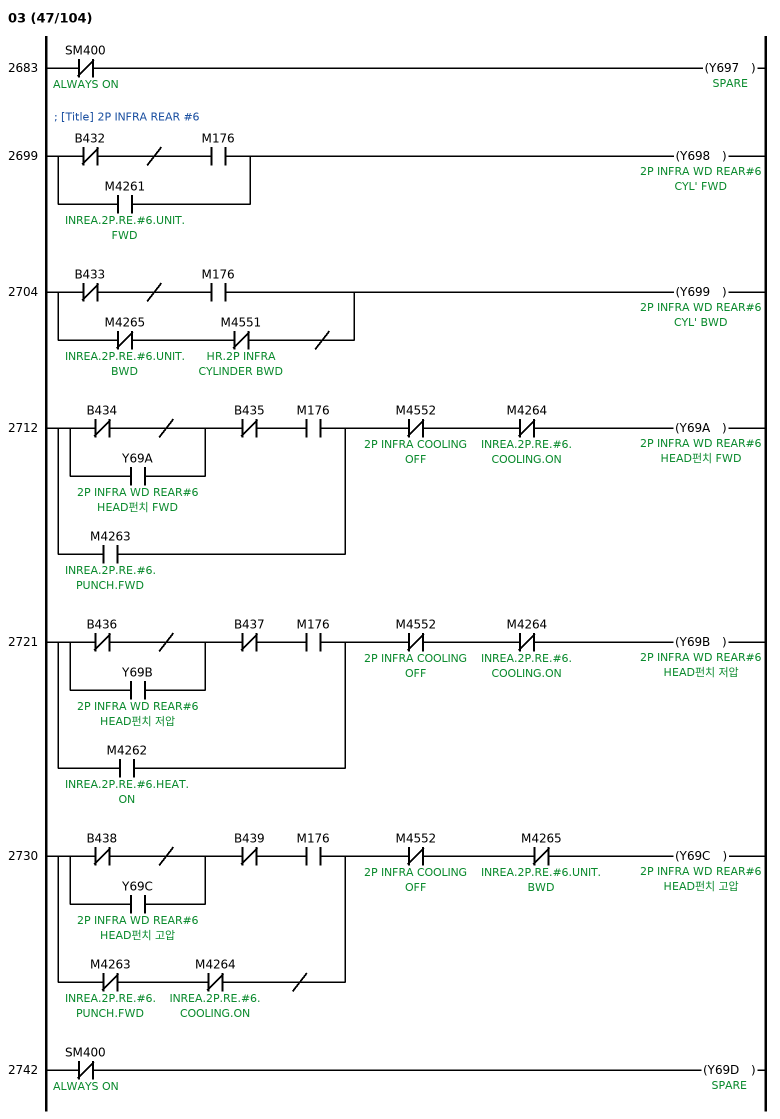
2683  LDI     SM400  ; ALWAYS ON
      OUT     Y697  ; SPARE
; [Title] 2P INFRA REAR #6
2699  LDI     B432
      INV
      AND     M176
      OR      M4261  ; INREA.2P.RE.#6.UNIT.FWD
      OUT     Y698  ; 2P INFRA WD REAR#6 CYL' FWD
2704  LDI     B433
      INV
      AND     M176
      LDI     M4265  ; INREA.2P.RE.#6.UNIT.BWD
      ANI     M4551  ; HR.2P INFRA CYLINDER BWD
      INV
      ORB
      OUT     Y699  ; 2P INFRA WD REAR#6 CYL' BWD
2712  LDI     B434
      INV
      OR      Y69A  ; 2P INFRA WD REAR#6 HEAD펀치 FWD
      ANI     B435
      AND     M176
      OR      M4263  ; INREA.2P.RE.#6.PUNCH.FWD
      ANI     M4552  ; 2P INFRA COOLING OFF
      ANI     M4264  ; INREA.2P.RE.#6.COOLING.ON
      OUT     Y69A  ; 2P INFRA WD REAR#6 HEAD펀치 FWD
2721  LDI     B436
      INV
      OR      Y69B  ; 2P INFRA WD REAR#6 HEAD펀치 저압
      ANI     B437
      AND     M176
      OR      M4262  ; INREA.2P.RE.#6.HEAT.ON
      ANI     M4552  ; 2P INFRA COOLING OFF
      ANI     M4264  ; INREA.2P.RE.#6.COOLING.ON
      OUT     Y69B  ; 2P INFRA WD REAR#6 HEAD펀치 저압
2730  LDI     B438
      INV
      OR      Y69C  ; 2P INFRA WD REAR#6 HEAD펀치 고압
      ANI     B439
      AND     M176
      LDI     M4263  ; INREA.2P.RE.#6.PUNCH.FWD
      ANI     M4264  ; INREA.2P.RE.#6.COOLING.ON
      INV
      ORB
      ANI     M4552  ; 2P INFRA COOLING OFF
      ANI     M4265  ; INREA.2P.RE.#6.UNIT.BWD
      OUT     Y69C  ; 2P INFRA WD REAR#6 HEAD펀치 고압
2742  LDI     SM400  ; ALWAYS ON
      OUT     Y69D  ; SPARE
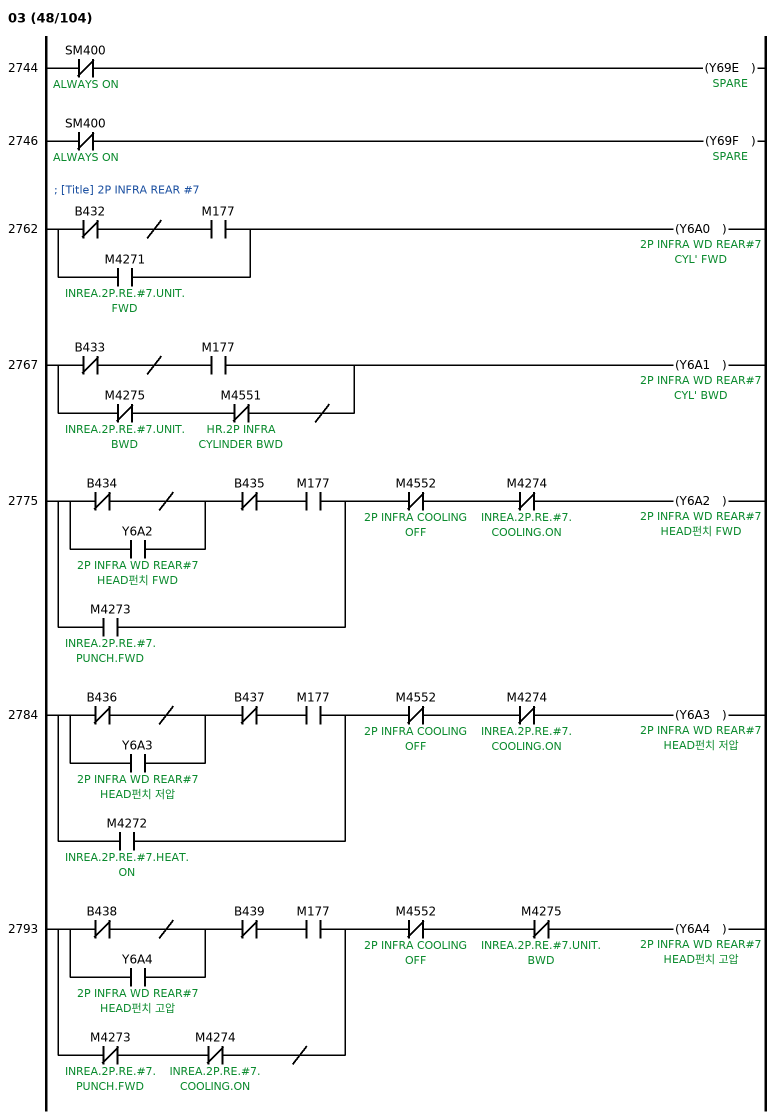
2744  LDI     SM400  ; ALWAYS ON
      OUT     Y69E  ; SPARE
2746  LDI     SM400  ; ALWAYS ON
      OUT     Y69F  ; SPARE
; [Title] 2P INFRA REAR #7
2762  LDI     B432
      INV
      AND     M177
      OR      M4271  ; INREA.2P.RE.#7.UNIT.FWD
      OUT     Y6A0  ; 2P INFRA WD REAR#7 CYL' FWD
2767  LDI     B433
      INV
      AND     M177
      LDI     M4275  ; INREA.2P.RE.#7.UNIT.BWD
      ANI     M4551  ; HR.2P INFRA CYLINDER BWD
      INV
      ORB
      OUT     Y6A1  ; 2P INFRA WD REAR#7 CYL' BWD
2775  LDI     B434
      INV
      OR      Y6A2  ; 2P INFRA WD REAR#7 HEAD펀치 FWD
      ANI     B435
      AND     M177
      OR      M4273  ; INREA.2P.RE.#7.PUNCH.FWD
      ANI     M4552  ; 2P INFRA COOLING OFF
      ANI     M4274  ; INREA.2P.RE.#7.COOLING.ON
      OUT     Y6A2  ; 2P INFRA WD REAR#7 HEAD펀치 FWD
2784  LDI     B436
      INV
      OR      Y6A3  ; 2P INFRA WD REAR#7 HEAD펀치 저압
      ANI     B437
      AND     M177
      OR      M4272  ; INREA.2P.RE.#7.HEAT.ON
      ANI     M4552  ; 2P INFRA COOLING OFF
      ANI     M4274  ; INREA.2P.RE.#7.COOLING.ON
      OUT     Y6A3  ; 2P INFRA WD REAR#7 HEAD펀치 저압
2793  LDI     B438
      INV
      OR      Y6A4  ; 2P INFRA WD REAR#7 HEAD펀치 고압
      ANI     B439
      AND     M177
      LDI     M4273  ; INREA.2P.RE.#7.PUNCH.FWD
      ANI     M4274  ; INREA.2P.RE.#7.COOLING.ON
      INV
      ORB
      ANI     M4552  ; 2P INFRA COOLING OFF
      ANI     M4275  ; INREA.2P.RE.#7.UNIT.BWD
      OUT     Y6A4  ; 2P INFRA WD REAR#7 HEAD펀치 고압
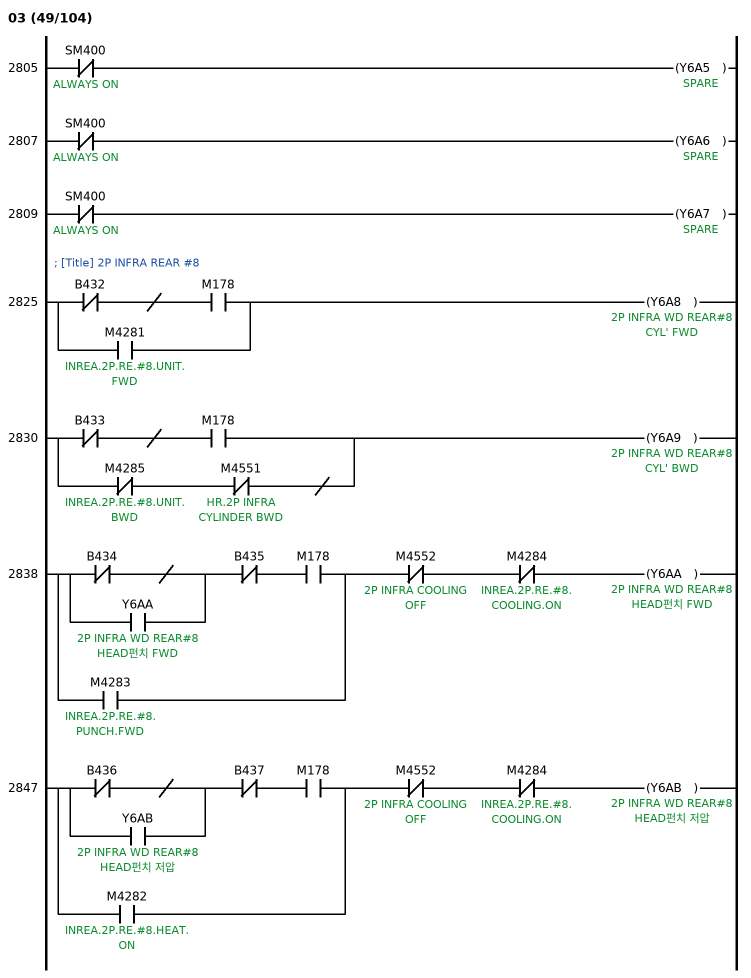
2805  LDI     SM400  ; ALWAYS ON
      OUT     Y6A5  ; SPARE
2807  LDI     SM400  ; ALWAYS ON
      OUT     Y6A6  ; SPARE
2809  LDI     SM400  ; ALWAYS ON
      OUT     Y6A7  ; SPARE
; [Title] 2P INFRA REAR #8
2825  LDI     B432
      INV
      AND     M178
      OR      M4281  ; INREA.2P.RE.#8.UNIT.FWD
      OUT     Y6A8  ; 2P INFRA WD REAR#8 CYL' FWD
2830  LDI     B433
      INV
      AND     M178
      LDI     M4285  ; INREA.2P.RE.#8.UNIT.BWD
      ANI     M4551  ; HR.2P INFRA CYLINDER BWD
      INV
      ORB
      OUT     Y6A9  ; 2P INFRA WD REAR#8 CYL' BWD
2838  LDI     B434
      INV
      OR      Y6AA  ; 2P INFRA WD REAR#8 HEAD펀치 FWD
      ANI     B435
      AND     M178
      OR      M4283  ; INREA.2P.RE.#8.PUNCH.FWD
      ANI     M4552  ; 2P INFRA COOLING OFF
      ANI     M4284  ; INREA.2P.RE.#8.COOLING.ON
      OUT     Y6AA  ; 2P INFRA WD REAR#8 HEAD펀치 FWD
2847  LDI     B436
      INV
      OR      Y6AB  ; 2P INFRA WD REAR#8 HEAD펀치 저압
      ANI     B437
      AND     M178
      OR      M4282  ; INREA.2P.RE.#8.HEAT.ON
      ANI     M4552  ; 2P INFRA COOLING OFF
      ANI     M4284  ; INREA.2P.RE.#8.COOLING.ON
      OUT     Y6AB  ; 2P INFRA WD REAR#8 HEAD펀치 저압
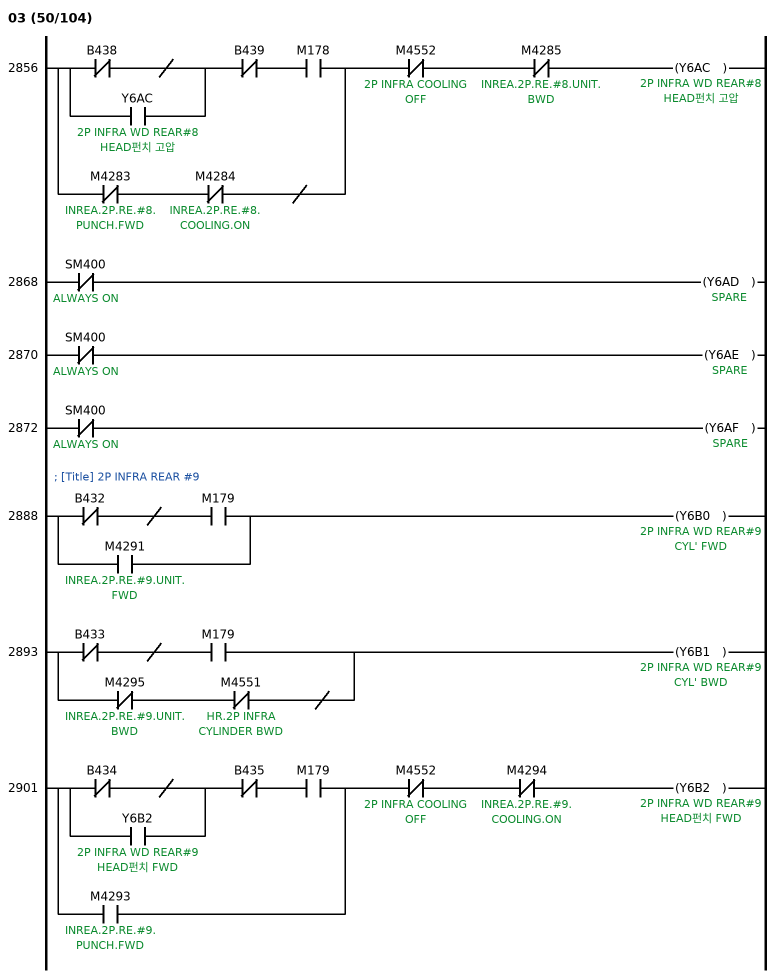
2856  LDI     B438
      INV
      OR      Y6AC  ; 2P INFRA WD REAR#8 HEAD펀치 고압
      ANI     B439
      AND     M178
      LDI     M4283  ; INREA.2P.RE.#8.PUNCH.FWD
      ANI     M4284  ; INREA.2P.RE.#8.COOLING.ON
      INV
      ORB
      ANI     M4552  ; 2P INFRA COOLING OFF
      ANI     M4285  ; INREA.2P.RE.#8.UNIT.BWD
      OUT     Y6AC  ; 2P INFRA WD REAR#8 HEAD펀치 고압
2868  LDI     SM400  ; ALWAYS ON
      OUT     Y6AD  ; SPARE
2870  LDI     SM400  ; ALWAYS ON
      OUT     Y6AE  ; SPARE
2872  LDI     SM400  ; ALWAYS ON
      OUT     Y6AF  ; SPARE
; [Title] 2P INFRA REAR #9
2888  LDI     B432
      INV
      AND     M179
      OR      M4291  ; INREA.2P.RE.#9.UNIT.FWD
      OUT     Y6B0  ; 2P INFRA WD REAR#9 CYL' FWD
2893  LDI     B433
      INV
      AND     M179
      LDI     M4295  ; INREA.2P.RE.#9.UNIT.BWD
      ANI     M4551  ; HR.2P INFRA CYLINDER BWD
      INV
      ORB
      OUT     Y6B1  ; 2P INFRA WD REAR#9 CYL' BWD
2901  LDI     B434
      INV
      OR      Y6B2  ; 2P INFRA WD REAR#9 HEAD펀치 FWD
      ANI     B435
      AND     M179
      OR      M4293  ; INREA.2P.RE.#9.PUNCH.FWD
      ANI     M4552  ; 2P INFRA COOLING OFF
      ANI     M4294  ; INREA.2P.RE.#9.COOLING.ON
      OUT     Y6B2  ; 2P INFRA WD REAR#9 HEAD펀치 FWD
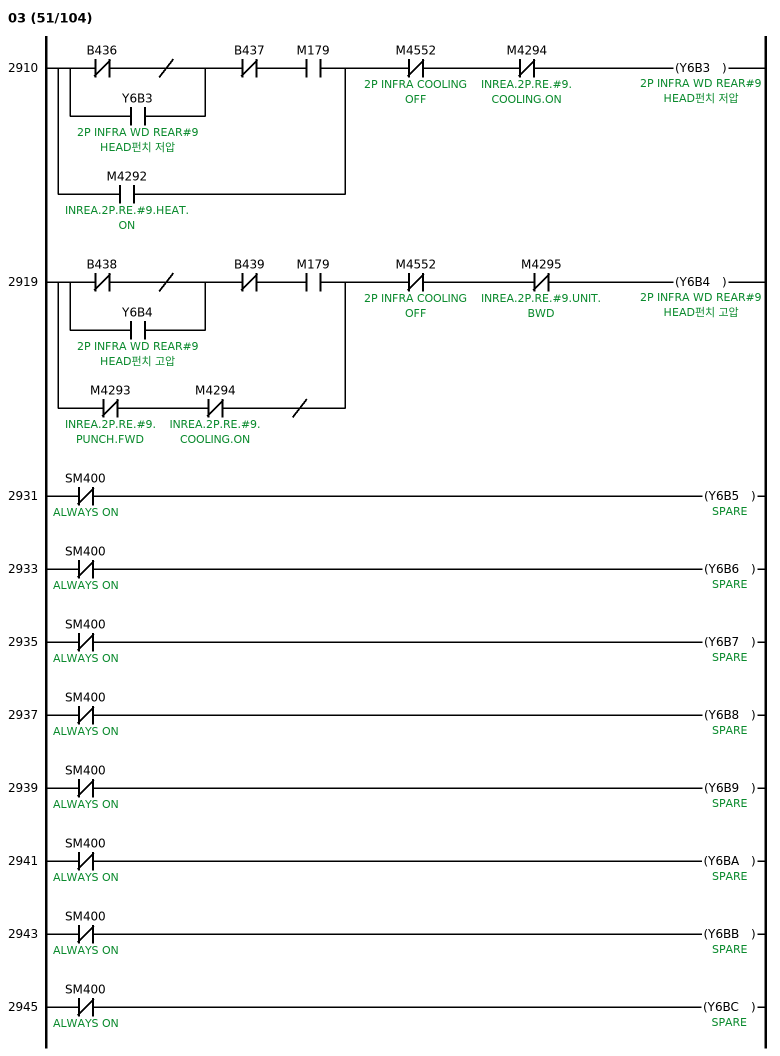
2910  LDI     B436
      INV
      OR      Y6B3  ; 2P INFRA WD REAR#9 HEAD펀치 저압
      ANI     B437
      AND     M179
      OR      M4292  ; INREA.2P.RE.#9.HEAT.ON
      ANI     M4552  ; 2P INFRA COOLING OFF
      ANI     M4294  ; INREA.2P.RE.#9.COOLING.ON
      OUT     Y6B3  ; 2P INFRA WD REAR#9 HEAD펀치 저압
2919  LDI     B438
      INV
      OR      Y6B4  ; 2P INFRA WD REAR#9 HEAD펀치 고압
      ANI     B439
      AND     M179
      LDI     M4293  ; INREA.2P.RE.#9.PUNCH.FWD
      ANI     M4294  ; INREA.2P.RE.#9.COOLING.ON
      INV
      ORB
      ANI     M4552  ; 2P INFRA COOLING OFF
      ANI     M4295  ; INREA.2P.RE.#9.UNIT.BWD
      OUT     Y6B4  ; 2P INFRA WD REAR#9 HEAD펀치 고압
2931  LDI     SM400  ; ALWAYS ON
      OUT     Y6B5  ; SPARE
2933  LDI     SM400  ; ALWAYS ON
      OUT     Y6B6  ; SPARE
2935  LDI     SM400  ; ALWAYS ON
      OUT     Y6B7  ; SPARE
2937  LDI     SM400  ; ALWAYS ON
      OUT     Y6B8  ; SPARE
2939  LDI     SM400  ; ALWAYS ON
      OUT     Y6B9  ; SPARE
2941  LDI     SM400  ; ALWAYS ON
      OUT     Y6BA  ; SPARE
2943  LDI     SM400  ; ALWAYS ON
      OUT     Y6BB  ; SPARE
2945  LDI     SM400  ; ALWAYS ON
      OUT     Y6BC  ; SPARE
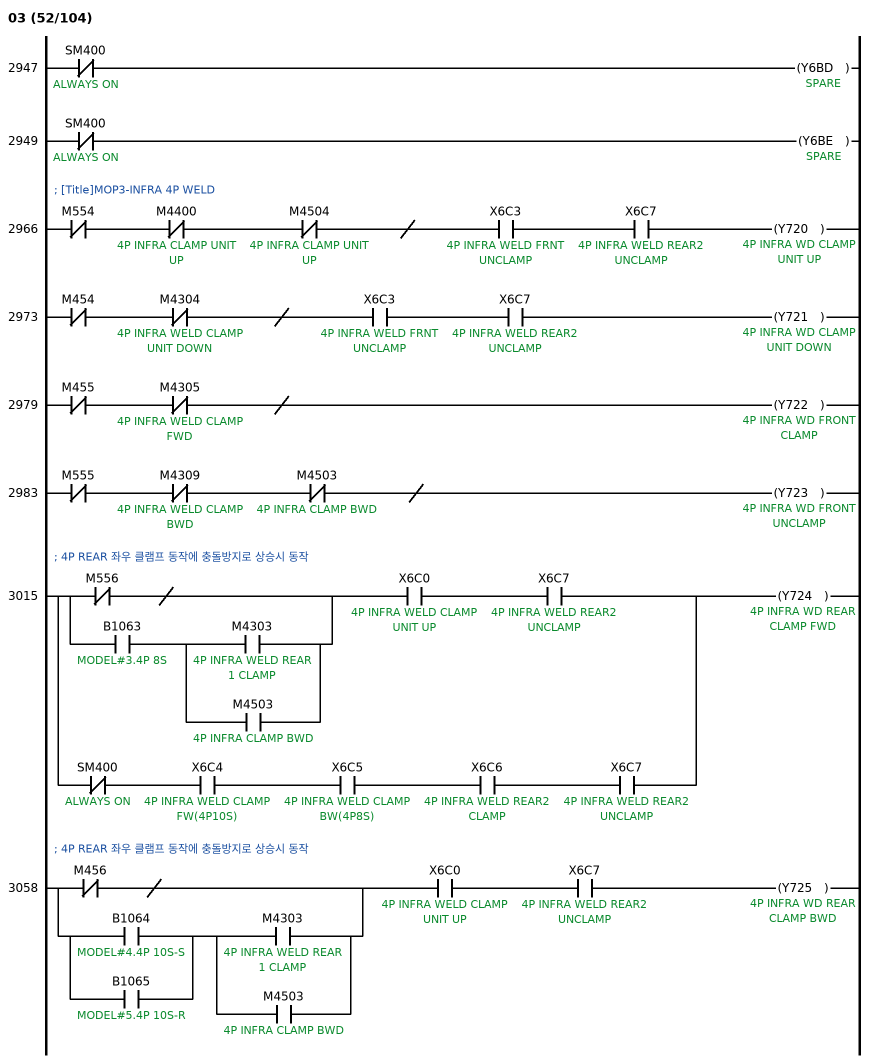
2947  LDI     SM400  ; ALWAYS ON
      OUT     Y6BD  ; SPARE
2949  LDI     SM400  ; ALWAYS ON
      OUT     Y6BE  ; SPARE
; [Title]MOP3-INFRA 4P WELD
2966  LDI     M554
      ANI     M4400  ; 4P INFRA CLAMP UNIT UP
      ANI     M4504  ; 4P INFRA CLAMP UNIT UP
      INV
      AND     X6C3  ; 4P INFRA WELD FRNT UNCLAMP
      AND     X6C7  ; 4P INFRA WELD REAR2 UNCLAMP
      OUT     Y720  ; 4P INFRA WD CLAMP UNIT UP
2973  LDI     M454
      ANI     M4304  ; 4P INFRA WELD CLAMP UNIT DOWN
      INV
      AND     X6C3  ; 4P INFRA WELD FRNT UNCLAMP
      AND     X6C7  ; 4P INFRA WELD REAR2 UNCLAMP
      OUT     Y721  ; 4P INFRA WD CLAMP UNIT DOWN
2979  LDI     M455
      ANI     M4305  ; 4P INFRA WELD CLAMP FWD
      INV
      OUT     Y722  ; 4P INFRA WD FRONT CLAMP
2983  LDI     M555
      ANI     M4309  ; 4P INFRA WELD CLAMP BWD
      ANI     M4503  ; 4P INFRA CLAMP BWD
      INV
      OUT     Y723  ; 4P INFRA WD FRONT UNCLAMP
; 4P REAR 좌우 클램프 동작에 충돌방지로 상승시 동작
3015  LDI     M556
      INV
      LD      B1063  ; MODEL#3.4P 8S
      LD      M4303  ; 4P INFRA WELD REAR 1 CLAMP
      OR      M4503  ; 4P INFRA CLAMP BWD
      ANB
      ORB
      AND     X6C0  ; 4P INFRA WELD CLAMP UNIT UP
      AND     X6C7  ; 4P INFRA WELD REAR2 UNCLAMP
      LDI     SM400  ; ALWAYS ON
      AND     X6C4  ; 4P INFRA WELD CLAMP FW(4P10S)
      AND     X6C5  ; 4P INFRA WELD CLAMP BW(4P8S)
      AND     X6C6  ; 4P INFRA WELD REAR2 CLAMP
      AND     X6C7  ; 4P INFRA WELD REAR2 UNCLAMP
      ORB
      OUT     Y724  ; 4P INFRA WD REAR CLAMP FWD
; 4P REAR 좌우 클램프 동작에 충돌방지로 상승시 동작
3058  LDI     M456
      INV
      LD      B1064  ; MODEL#4.4P 10S-S
      OR      B1065  ; MODEL#5.4P 10S-R
      LD      M4303  ; 4P INFRA WELD REAR 1 CLAMP
      OR      M4503  ; 4P INFRA CLAMP BWD
      ANB
      ORB
      AND     X6C0  ; 4P INFRA WELD CLAMP UNIT UP
      AND     X6C7  ; 4P INFRA WELD REAR2 UNCLAMP
      OUT     Y725  ; 4P INFRA WD REAR CLAMP BWD
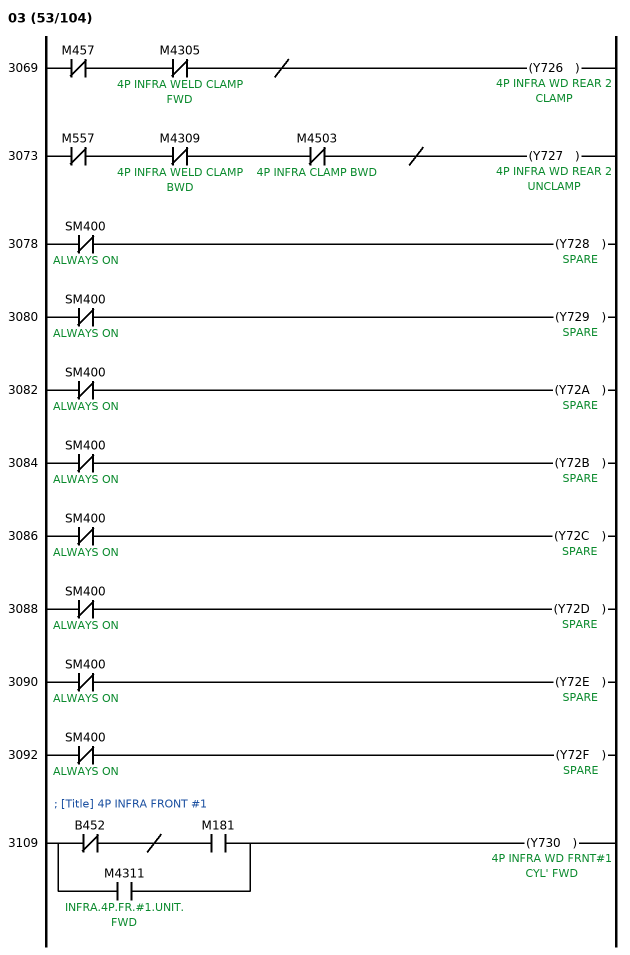
3069  LDI     M457
      ANI     M4305  ; 4P INFRA WELD CLAMP FWD
      INV
      OUT     Y726  ; 4P INFRA WD REAR 2 CLAMP
3073  LDI     M557
      ANI     M4309  ; 4P INFRA WELD CLAMP BWD
      ANI     M4503  ; 4P INFRA CLAMP BWD
      INV
      OUT     Y727  ; 4P INFRA WD REAR 2 UNCLAMP
3078  LDI     SM400  ; ALWAYS ON
      OUT     Y728  ; SPARE
3080  LDI     SM400  ; ALWAYS ON
      OUT     Y729  ; SPARE
3082  LDI     SM400  ; ALWAYS ON
      OUT     Y72A  ; SPARE
3084  LDI     SM400  ; ALWAYS ON
      OUT     Y72B  ; SPARE
3086  LDI     SM400  ; ALWAYS ON
      OUT     Y72C  ; SPARE
3088  LDI     SM400  ; ALWAYS ON
      OUT     Y72D  ; SPARE
3090  LDI     SM400  ; ALWAYS ON
      OUT     Y72E  ; SPARE
3092  LDI     SM400  ; ALWAYS ON
      OUT     Y72F  ; SPARE
; [Title] 4P INFRA FRONT #1
3109  LDI     B452
      INV
      AND     M181
      OR      M4311  ; INFRA.4P.FR.#1.UNIT.FWD
      OUT     Y730  ; 4P INFRA WD FRNT#1 CYL' FWD
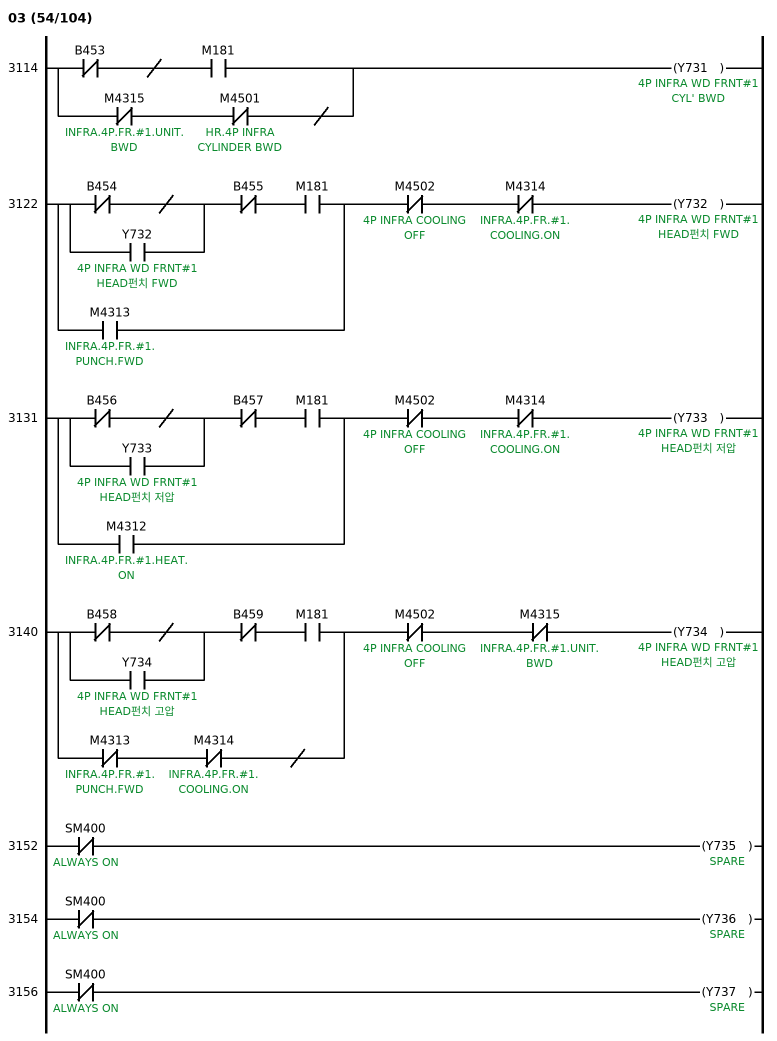
3114  LDI     B453
      INV
      AND     M181
      LDI     M4315  ; INFRA.4P.FR.#1.UNIT.BWD
      ANI     M4501  ; HR.4P INFRA CYLINDER BWD
      INV
      ORB
      OUT     Y731  ; 4P INFRA WD FRNT#1 CYL' BWD
3122  LDI     B454
      INV
      OR      Y732  ; 4P INFRA WD FRNT#1 HEAD펀치 FWD
      ANI     B455
      AND     M181
      OR      M4313  ; INFRA.4P.FR.#1.PUNCH.FWD
      ANI     M4502  ; 4P INFRA COOLING OFF
      ANI     M4314  ; INFRA.4P.FR.#1.COOLING.ON
      OUT     Y732  ; 4P INFRA WD FRNT#1 HEAD펀치 FWD
3131  LDI     B456
      INV
      OR      Y733  ; 4P INFRA WD FRNT#1 HEAD펀치 저압
      ANI     B457
      AND     M181
      OR      M4312  ; INFRA.4P.FR.#1.HEAT.ON
      ANI     M4502  ; 4P INFRA COOLING OFF
      ANI     M4314  ; INFRA.4P.FR.#1.COOLING.ON
      OUT     Y733  ; 4P INFRA WD FRNT#1 HEAD펀치 저압
3140  LDI     B458
      INV
      OR      Y734  ; 4P INFRA WD FRNT#1 HEAD펀치 고압
      ANI     B459
      AND     M181
      LDI     M4313  ; INFRA.4P.FR.#1.PUNCH.FWD
      ANI     M4314  ; INFRA.4P.FR.#1.COOLING.ON
      INV
      ORB
      ANI     M4502  ; 4P INFRA COOLING OFF
      ANI     M4315  ; INFRA.4P.FR.#1.UNIT.BWD
      OUT     Y734  ; 4P INFRA WD FRNT#1 HEAD펀치 고압
3152  LDI     SM400  ; ALWAYS ON
      OUT     Y735  ; SPARE
3154  LDI     SM400  ; ALWAYS ON
      OUT     Y736  ; SPARE
3156  LDI     SM400  ; ALWAYS ON
      OUT     Y737  ; SPARE
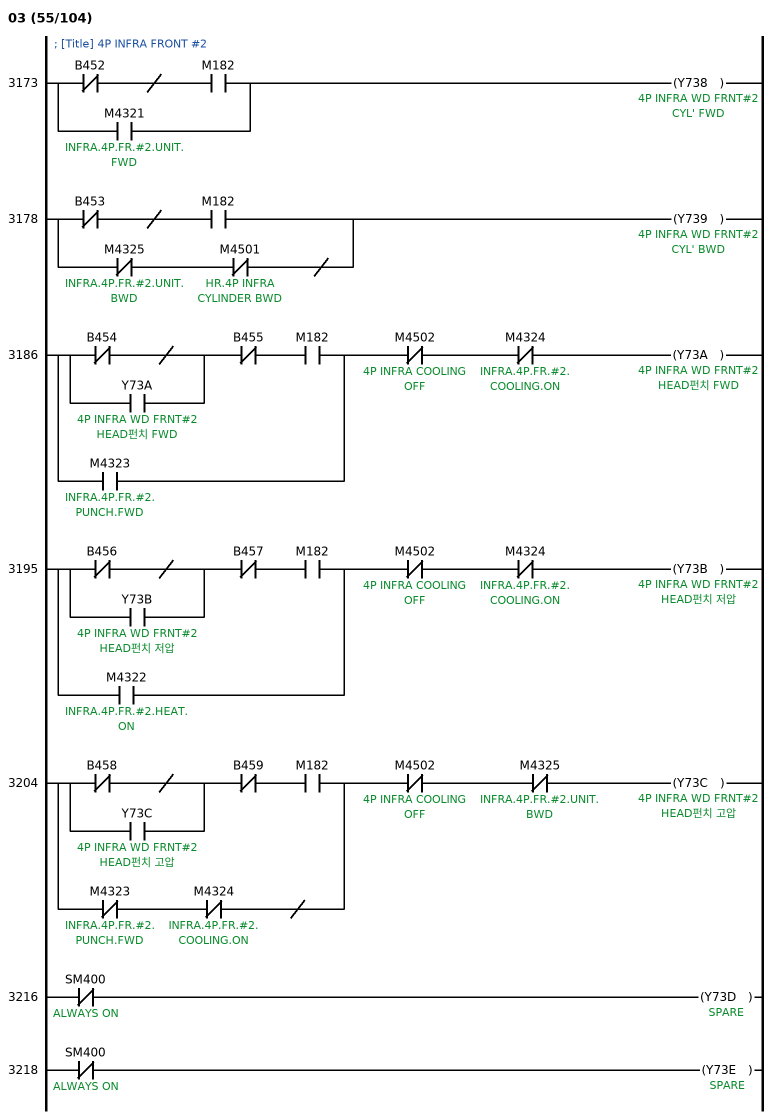
; [Title] 4P INFRA FRONT #2
3173  LDI     B452
      INV
      AND     M182
      OR      M4321  ; INFRA.4P.FR.#2.UNIT.FWD
      OUT     Y738  ; 4P INFRA WD FRNT#2 CYL' FWD
3178  LDI     B453
      INV
      AND     M182
      LDI     M4325  ; INFRA.4P.FR.#2.UNIT.BWD
      ANI     M4501  ; HR.4P INFRA CYLINDER BWD
      INV
      ORB
      OUT     Y739  ; 4P INFRA WD FRNT#2 CYL' BWD
3186  LDI     B454
      INV
      OR      Y73A  ; 4P INFRA WD FRNT#2 HEAD펀치 FWD
      ANI     B455
      AND     M182
      OR      M4323  ; INFRA.4P.FR.#2.PUNCH.FWD
      ANI     M4502  ; 4P INFRA COOLING OFF
      ANI     M4324  ; INFRA.4P.FR.#2.COOLING.ON
      OUT     Y73A  ; 4P INFRA WD FRNT#2 HEAD펀치 FWD
3195  LDI     B456
      INV
      OR      Y73B  ; 4P INFRA WD FRNT#2 HEAD펀치 저압
      ANI     B457
      AND     M182
      OR      M4322  ; INFRA.4P.FR.#2.HEAT.ON
      ANI     M4502  ; 4P INFRA COOLING OFF
      ANI     M4324  ; INFRA.4P.FR.#2.COOLING.ON
      OUT     Y73B  ; 4P INFRA WD FRNT#2 HEAD펀치 저압
3204  LDI     B458
      INV
      OR      Y73C  ; 4P INFRA WD FRNT#2 HEAD펀치 고압
      ANI     B459
      AND     M182
      LDI     M4323  ; INFRA.4P.FR.#2.PUNCH.FWD
      ANI     M4324  ; INFRA.4P.FR.#2.COOLING.ON
      INV
      ORB
      ANI     M4502  ; 4P INFRA COOLING OFF
      ANI     M4325  ; INFRA.4P.FR.#2.UNIT.BWD
      OUT     Y73C  ; 4P INFRA WD FRNT#2 HEAD펀치 고압
3216  LDI     SM400  ; ALWAYS ON
      OUT     Y73D  ; SPARE
3218  LDI     SM400  ; ALWAYS ON
      OUT     Y73E  ; SPARE
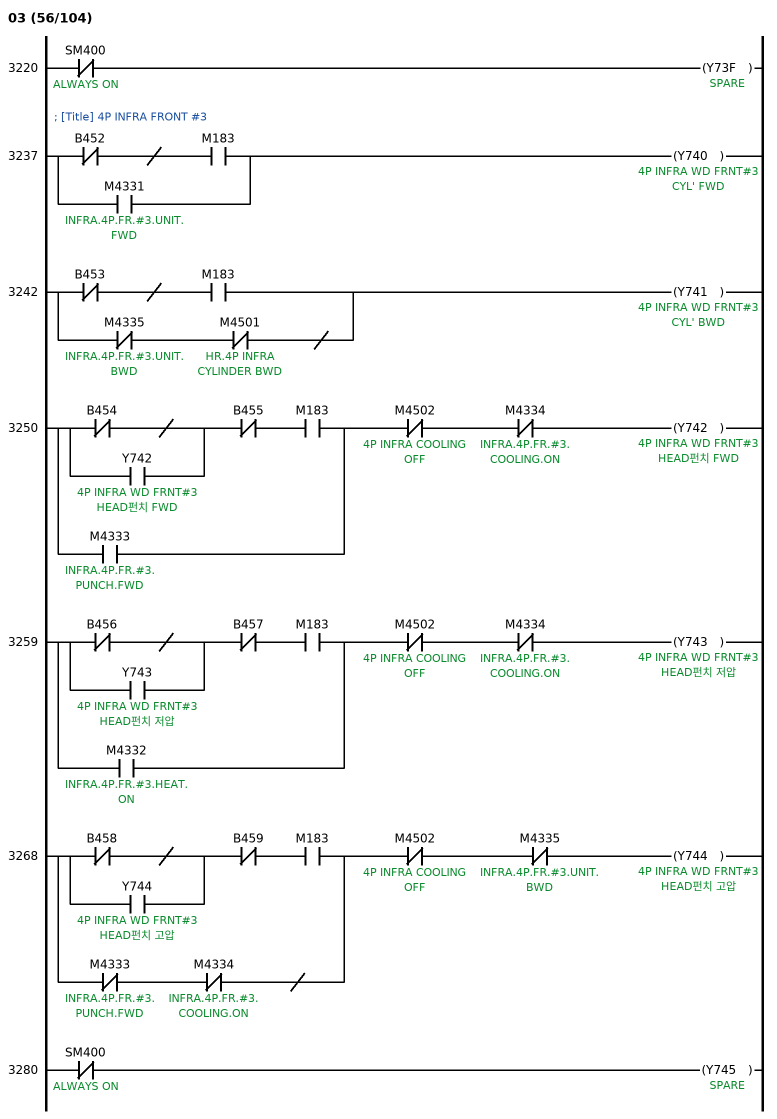
3220  LDI     SM400  ; ALWAYS ON
      OUT     Y73F  ; SPARE
; [Title] 4P INFRA FRONT #3
3237  LDI     B452
      INV
      AND     M183
      OR      M4331  ; INFRA.4P.FR.#3.UNIT.FWD
      OUT     Y740  ; 4P INFRA WD FRNT#3 CYL' FWD
3242  LDI     B453
      INV
      AND     M183
      LDI     M4335  ; INFRA.4P.FR.#3.UNIT.BWD
      ANI     M4501  ; HR.4P INFRA CYLINDER BWD
      INV
      ORB
      OUT     Y741  ; 4P INFRA WD FRNT#3 CYL' BWD
3250  LDI     B454
      INV
      OR      Y742  ; 4P INFRA WD FRNT#3 HEAD펀치 FWD
      ANI     B455
      AND     M183
      OR      M4333  ; INFRA.4P.FR.#3.PUNCH.FWD
      ANI     M4502  ; 4P INFRA COOLING OFF
      ANI     M4334  ; INFRA.4P.FR.#3.COOLING.ON
      OUT     Y742  ; 4P INFRA WD FRNT#3 HEAD펀치 FWD
3259  LDI     B456
      INV
      OR      Y743  ; 4P INFRA WD FRNT#3 HEAD펀치 저압
      ANI     B457
      AND     M183
      OR      M4332  ; INFRA.4P.FR.#3.HEAT.ON
      ANI     M4502  ; 4P INFRA COOLING OFF
      ANI     M4334  ; INFRA.4P.FR.#3.COOLING.ON
      OUT     Y743  ; 4P INFRA WD FRNT#3 HEAD펀치 저압
3268  LDI     B458
      INV
      OR      Y744  ; 4P INFRA WD FRNT#3 HEAD펀치 고압
      ANI     B459
      AND     M183
      LDI     M4333  ; INFRA.4P.FR.#3.PUNCH.FWD
      ANI     M4334  ; INFRA.4P.FR.#3.COOLING.ON
      INV
      ORB
      ANI     M4502  ; 4P INFRA COOLING OFF
      ANI     M4335  ; INFRA.4P.FR.#3.UNIT.BWD
      OUT     Y744  ; 4P INFRA WD FRNT#3 HEAD펀치 고압
3280  LDI     SM400  ; ALWAYS ON
      OUT     Y745  ; SPARE
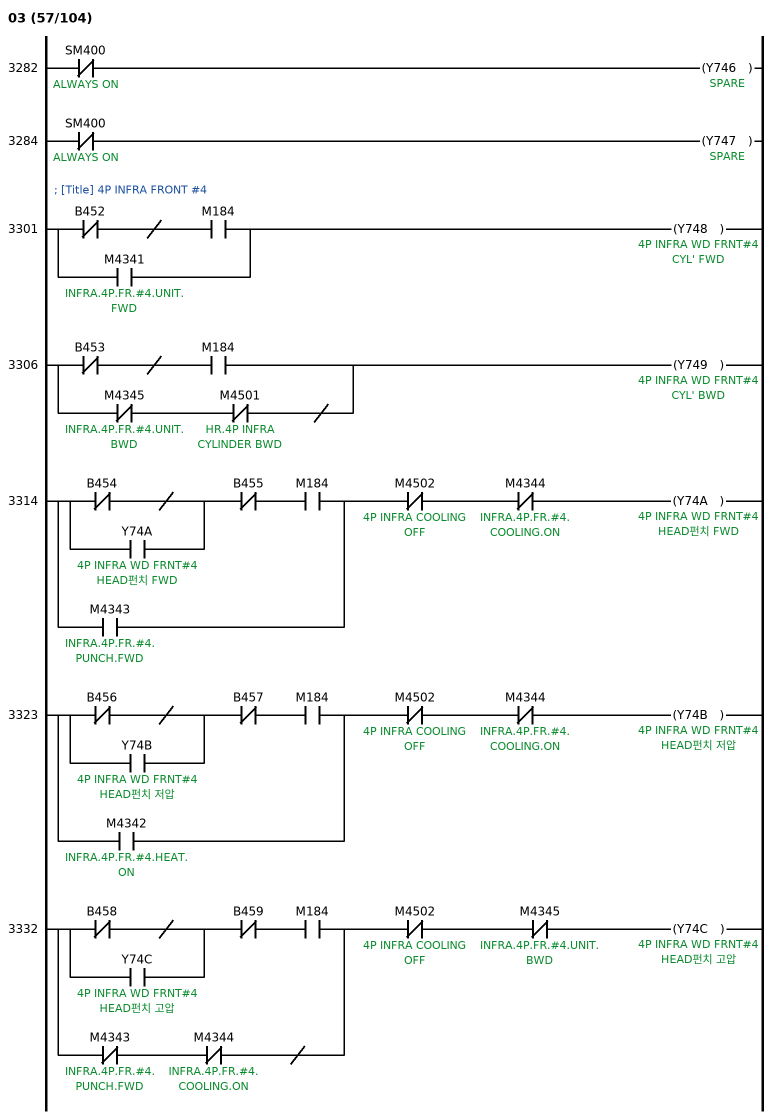
3282  LDI     SM400  ; ALWAYS ON
      OUT     Y746  ; SPARE
3284  LDI     SM400  ; ALWAYS ON
      OUT     Y747  ; SPARE
; [Title] 4P INFRA FRONT #4
3301  LDI     B452
      INV
      AND     M184
      OR      M4341  ; INFRA.4P.FR.#4.UNIT.FWD
      OUT     Y748  ; 4P INFRA WD FRNT#4 CYL' FWD
3306  LDI     B453
      INV
      AND     M184
      LDI     M4345  ; INFRA.4P.FR.#4.UNIT.BWD
      ANI     M4501  ; HR.4P INFRA CYLINDER BWD
      INV
      ORB
      OUT     Y749  ; 4P INFRA WD FRNT#4 CYL' BWD
3314  LDI     B454
      INV
      OR      Y74A  ; 4P INFRA WD FRNT#4 HEAD펀치 FWD
      ANI     B455
      AND     M184
      OR      M4343  ; INFRA.4P.FR.#4.PUNCH.FWD
      ANI     M4502  ; 4P INFRA COOLING OFF
      ANI     M4344  ; INFRA.4P.FR.#4.COOLING.ON
      OUT     Y74A  ; 4P INFRA WD FRNT#4 HEAD펀치 FWD
3323  LDI     B456
      INV
      OR      Y74B  ; 4P INFRA WD FRNT#4 HEAD펀치 저압
      ANI     B457
      AND     M184
      OR      M4342  ; INFRA.4P.FR.#4.HEAT.ON
      ANI     M4502  ; 4P INFRA COOLING OFF
      ANI     M4344  ; INFRA.4P.FR.#4.COOLING.ON
      OUT     Y74B  ; 4P INFRA WD FRNT#4 HEAD펀치 저압
3332  LDI     B458
      INV
      OR      Y74C  ; 4P INFRA WD FRNT#4 HEAD펀치 고압
      ANI     B459
      AND     M184
      LDI     M4343  ; INFRA.4P.FR.#4.PUNCH.FWD
      ANI     M4344  ; INFRA.4P.FR.#4.COOLING.ON
      INV
      ORB
      ANI     M4502  ; 4P INFRA COOLING OFF
      ANI     M4345  ; INFRA.4P.FR.#4.UNIT.BWD
      OUT     Y74C  ; 4P INFRA WD FRNT#4 HEAD펀치 고압
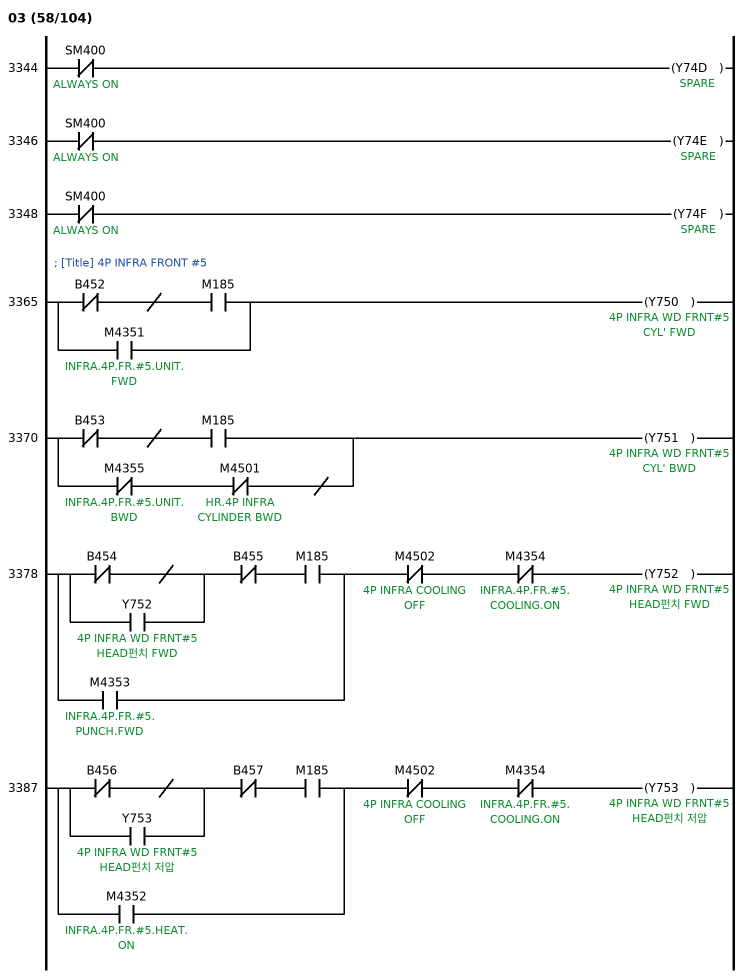
3344  LDI     SM400  ; ALWAYS ON
      OUT     Y74D  ; SPARE
3346  LDI     SM400  ; ALWAYS ON
      OUT     Y74E  ; SPARE
3348  LDI     SM400  ; ALWAYS ON
      OUT     Y74F  ; SPARE
; [Title] 4P INFRA FRONT #5
3365  LDI     B452
      INV
      AND     M185
      OR      M4351  ; INFRA.4P.FR.#5.UNIT.FWD
      OUT     Y750  ; 4P INFRA WD FRNT#5 CYL' FWD
3370  LDI     B453
      INV
      AND     M185
      LDI     M4355  ; INFRA.4P.FR.#5.UNIT.BWD
      ANI     M4501  ; HR.4P INFRA CYLINDER BWD
      INV
      ORB
      OUT     Y751  ; 4P INFRA WD FRNT#5 CYL' BWD
3378  LDI     B454
      INV
      OR      Y752  ; 4P INFRA WD FRNT#5 HEAD펀치 FWD
      ANI     B455
      AND     M185
      OR      M4353  ; INFRA.4P.FR.#5.PUNCH.FWD
      ANI     M4502  ; 4P INFRA COOLING OFF
      ANI     M4354  ; INFRA.4P.FR.#5.COOLING.ON
      OUT     Y752  ; 4P INFRA WD FRNT#5 HEAD펀치 FWD
3387  LDI     B456
      INV
      OR      Y753  ; 4P INFRA WD FRNT#5 HEAD펀치 저압
      ANI     B457
      AND     M185
      OR      M4352  ; INFRA.4P.FR.#5.HEAT.ON
      ANI     M4502  ; 4P INFRA COOLING OFF
      ANI     M4354  ; INFRA.4P.FR.#5.COOLING.ON
      OUT     Y753  ; 4P INFRA WD FRNT#5 HEAD펀치 저압
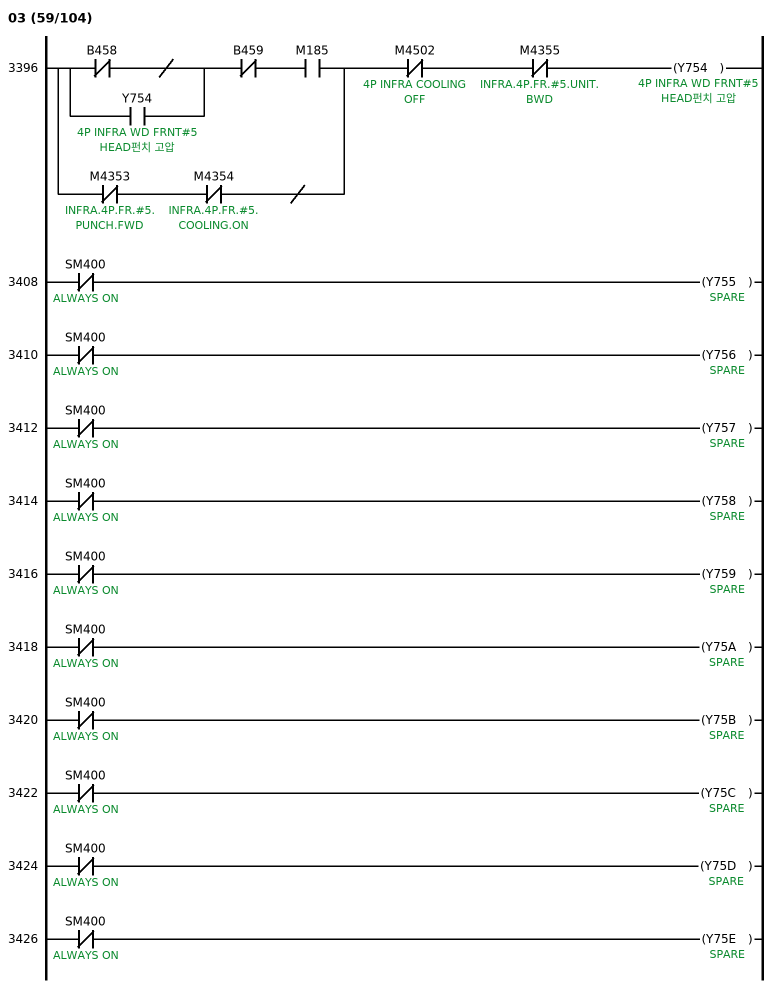
3396  LDI     B458
      INV
      OR      Y754  ; 4P INFRA WD FRNT#5 HEAD펀치 고압
      ANI     B459
      AND     M185
      LDI     M4353  ; INFRA.4P.FR.#5.PUNCH.FWD
      ANI     M4354  ; INFRA.4P.FR.#5.COOLING.ON
      INV
      ORB
      ANI     M4502  ; 4P INFRA COOLING OFF
      ANI     M4355  ; INFRA.4P.FR.#5.UNIT.BWD
      OUT     Y754  ; 4P INFRA WD FRNT#5 HEAD펀치 고압
3408  LDI     SM400  ; ALWAYS ON
      OUT     Y755  ; SPARE
3410  LDI     SM400  ; ALWAYS ON
      OUT     Y756  ; SPARE
3412  LDI     SM400  ; ALWAYS ON
      OUT     Y757  ; SPARE
3414  LDI     SM400  ; ALWAYS ON
      OUT     Y758  ; SPARE
3416  LDI     SM400  ; ALWAYS ON
      OUT     Y759  ; SPARE
3418  LDI     SM400  ; ALWAYS ON
      OUT     Y75A  ; SPARE
3420  LDI     SM400  ; ALWAYS ON
      OUT     Y75B  ; SPARE
3422  LDI     SM400  ; ALWAYS ON
      OUT     Y75C  ; SPARE
3424  LDI     SM400  ; ALWAYS ON
      OUT     Y75D  ; SPARE
3426  LDI     SM400  ; ALWAYS ON
      OUT     Y75E  ; SPARE
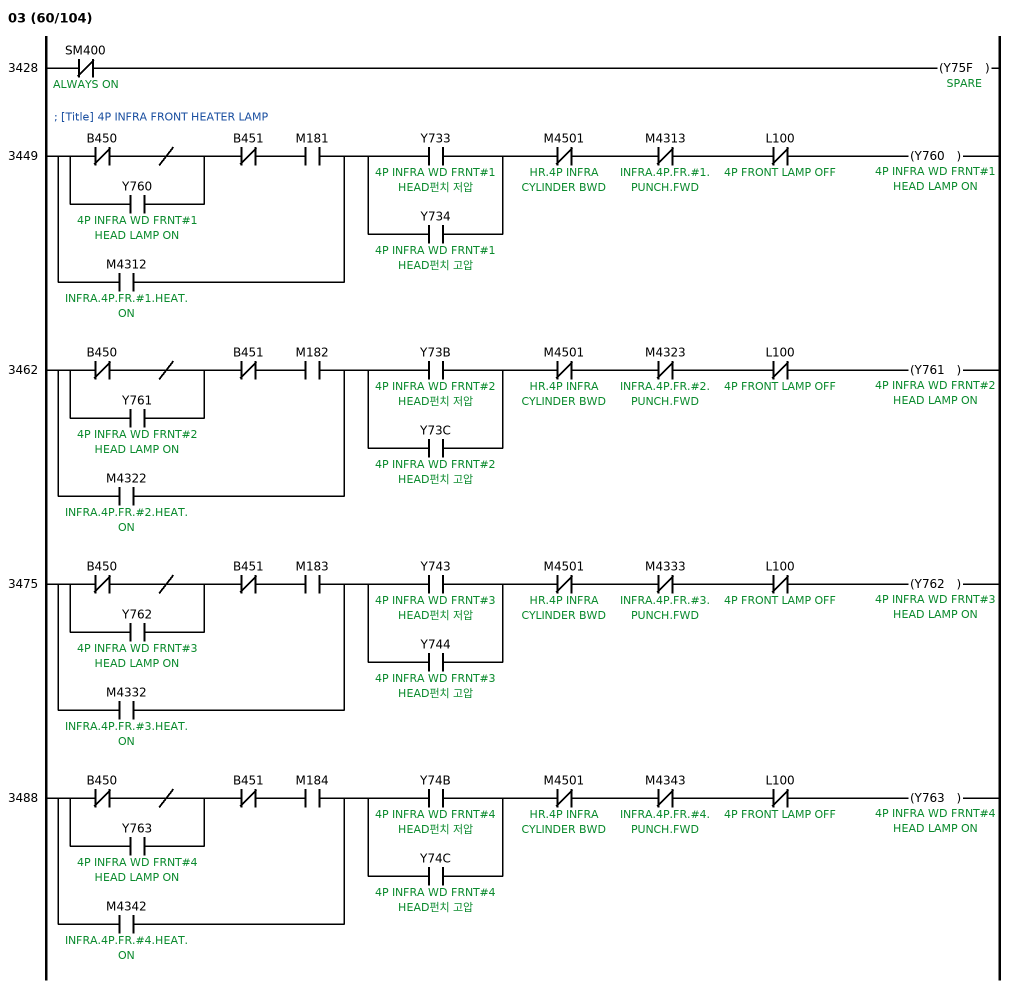
3428  LDI     SM400  ; ALWAYS ON
      OUT     Y75F  ; SPARE
; [Title] 4P INFRA FRONT HEATER LAMP
3449  LDI     B450
      INV
      OR      Y760  ; 4P INFRA WD FRNT#1 HEAD LAMP ON
      ANI     B451
      AND     M181
      OR      M4312  ; INFRA.4P.FR.#1.HEAT.ON
      LD      Y733  ; 4P INFRA WD FRNT#1 HEAD펀치 저압
      OR      Y734  ; 4P INFRA WD FRNT#1 HEAD펀치 고압
      ANB
      ANI     M4501  ; HR.4P INFRA CYLINDER BWD
      ANI     M4313  ; INFRA.4P.FR.#1.PUNCH.FWD
      ANI     L100  ; 4P FRONT LAMP OFF
      OUT     Y760  ; 4P INFRA WD FRNT#1 HEAD LAMP ON
3462  LDI     B450
      INV
      OR      Y761  ; 4P INFRA WD FRNT#2 HEAD LAMP ON
      ANI     B451
      AND     M182
      OR      M4322  ; INFRA.4P.FR.#2.HEAT.ON
      LD      Y73B  ; 4P INFRA WD FRNT#2 HEAD펀치 저압
      OR      Y73C  ; 4P INFRA WD FRNT#2 HEAD펀치 고압
      ANB
      ANI     M4501  ; HR.4P INFRA CYLINDER BWD
      ANI     M4323  ; INFRA.4P.FR.#2.PUNCH.FWD
      ANI     L100  ; 4P FRONT LAMP OFF
      OUT     Y761  ; 4P INFRA WD FRNT#2 HEAD LAMP ON
3475  LDI     B450
      INV
      OR      Y762  ; 4P INFRA WD FRNT#3 HEAD LAMP ON
      ANI     B451
      AND     M183
      OR      M4332  ; INFRA.4P.FR.#3.HEAT.ON
      LD      Y743  ; 4P INFRA WD FRNT#3 HEAD펀치 저압
      OR      Y744  ; 4P INFRA WD FRNT#3 HEAD펀치 고압
      ANB
      ANI     M4501  ; HR.4P INFRA CYLINDER BWD
      ANI     M4333  ; INFRA.4P.FR.#3.PUNCH.FWD
      ANI     L100  ; 4P FRONT LAMP OFF
      OUT     Y762  ; 4P INFRA WD FRNT#3 HEAD LAMP ON
3488  LDI     B450
      INV
      OR      Y763  ; 4P INFRA WD FRNT#4 HEAD LAMP ON
      ANI     B451
      AND     M184
      OR      M4342  ; INFRA.4P.FR.#4.HEAT.ON
      LD      Y74B  ; 4P INFRA WD FRNT#4 HEAD펀치 저압
      OR      Y74C  ; 4P INFRA WD FRNT#4 HEAD펀치 고압
      ANB
      ANI     M4501  ; HR.4P INFRA CYLINDER BWD
      ANI     M4343  ; INFRA.4P.FR.#4.PUNCH.FWD
      ANI     L100  ; 4P FRONT LAMP OFF
      OUT     Y763  ; 4P INFRA WD FRNT#4 HEAD LAMP ON
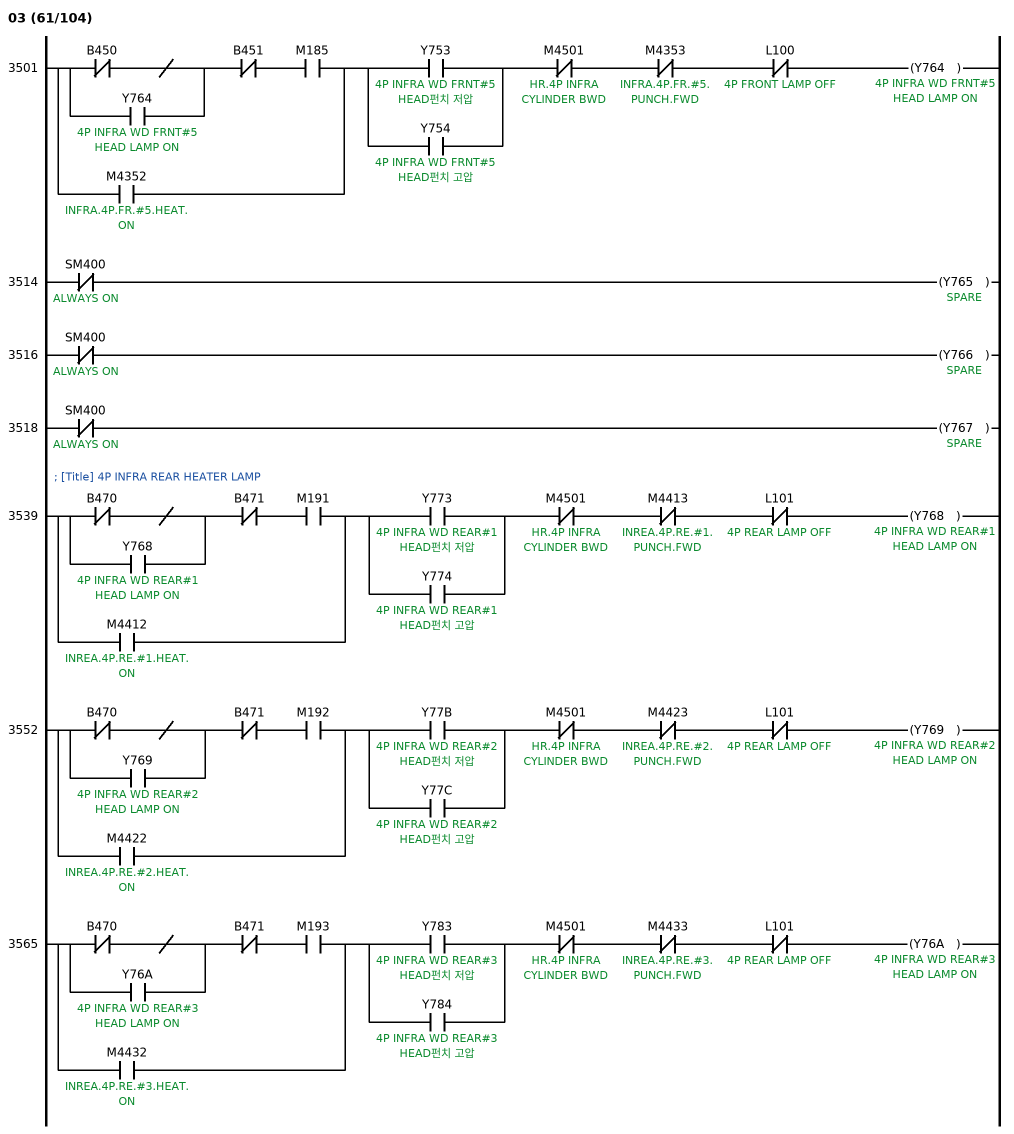
3501  LDI     B450
      INV
      OR      Y764  ; 4P INFRA WD FRNT#5 HEAD LAMP ON
      ANI     B451
      AND     M185
      OR      M4352  ; INFRA.4P.FR.#5.HEAT.ON
      LD      Y753  ; 4P INFRA WD FRNT#5 HEAD펀치 저압
      OR      Y754  ; 4P INFRA WD FRNT#5 HEAD펀치 고압
      ANB
      ANI     M4501  ; HR.4P INFRA CYLINDER BWD
      ANI     M4353  ; INFRA.4P.FR.#5.PUNCH.FWD
      ANI     L100  ; 4P FRONT LAMP OFF
      OUT     Y764  ; 4P INFRA WD FRNT#5 HEAD LAMP ON
3514  LDI     SM400  ; ALWAYS ON
      OUT     Y765  ; SPARE
3516  LDI     SM400  ; ALWAYS ON
      OUT     Y766  ; SPARE
3518  LDI     SM400  ; ALWAYS ON
      OUT     Y767  ; SPARE
; [Title] 4P INFRA REAR HEATER LAMP
3539  LDI     B470
      INV
      OR      Y768  ; 4P INFRA WD REAR#1 HEAD LAMP ON
      ANI     B471
      AND     M191
      OR      M4412  ; INREA.4P.RE.#1.HEAT.ON
      LD      Y773  ; 4P INFRA WD REAR#1 HEAD펀치 저압
      OR      Y774  ; 4P INFRA WD REAR#1 HEAD펀치 고압
      ANB
      ANI     M4501  ; HR.4P INFRA CYLINDER BWD
      ANI     M4413  ; INREA.4P.RE.#1.PUNCH.FWD
      ANI     L101  ; 4P REAR LAMP OFF
      OUT     Y768  ; 4P INFRA WD REAR#1 HEAD LAMP ON
3552  LDI     B470
      INV
      OR      Y769  ; 4P INFRA WD REAR#2 HEAD LAMP ON
      ANI     B471
      AND     M192
      OR      M4422  ; INREA.4P.RE.#2.HEAT.ON
      LD      Y77B  ; 4P INFRA WD REAR#2 HEAD펀치 저압
      OR      Y77C  ; 4P INFRA WD REAR#2 HEAD펀치 고압
      ANB
      ANI     M4501  ; HR.4P INFRA CYLINDER BWD
      ANI     M4423  ; INREA.4P.RE.#2.PUNCH.FWD
      ANI     L101  ; 4P REAR LAMP OFF
      OUT     Y769  ; 4P INFRA WD REAR#2 HEAD LAMP ON
3565  LDI     B470
      INV
      OR      Y76A  ; 4P INFRA WD REAR#3 HEAD LAMP ON
      ANI     B471
      AND     M193
      OR      M4432  ; INREA.4P.RE.#3.HEAT.ON
      LD      Y783  ; 4P INFRA WD REAR#3 HEAD펀치 저압
      OR      Y784  ; 4P INFRA WD REAR#3 HEAD펀치 고압
      ANB
      ANI     M4501  ; HR.4P INFRA CYLINDER BWD
      ANI     M4433  ; INREA.4P.RE.#3.PUNCH.FWD
      ANI     L101  ; 4P REAR LAMP OFF
      OUT     Y76A  ; 4P INFRA WD REAR#3 HEAD LAMP ON
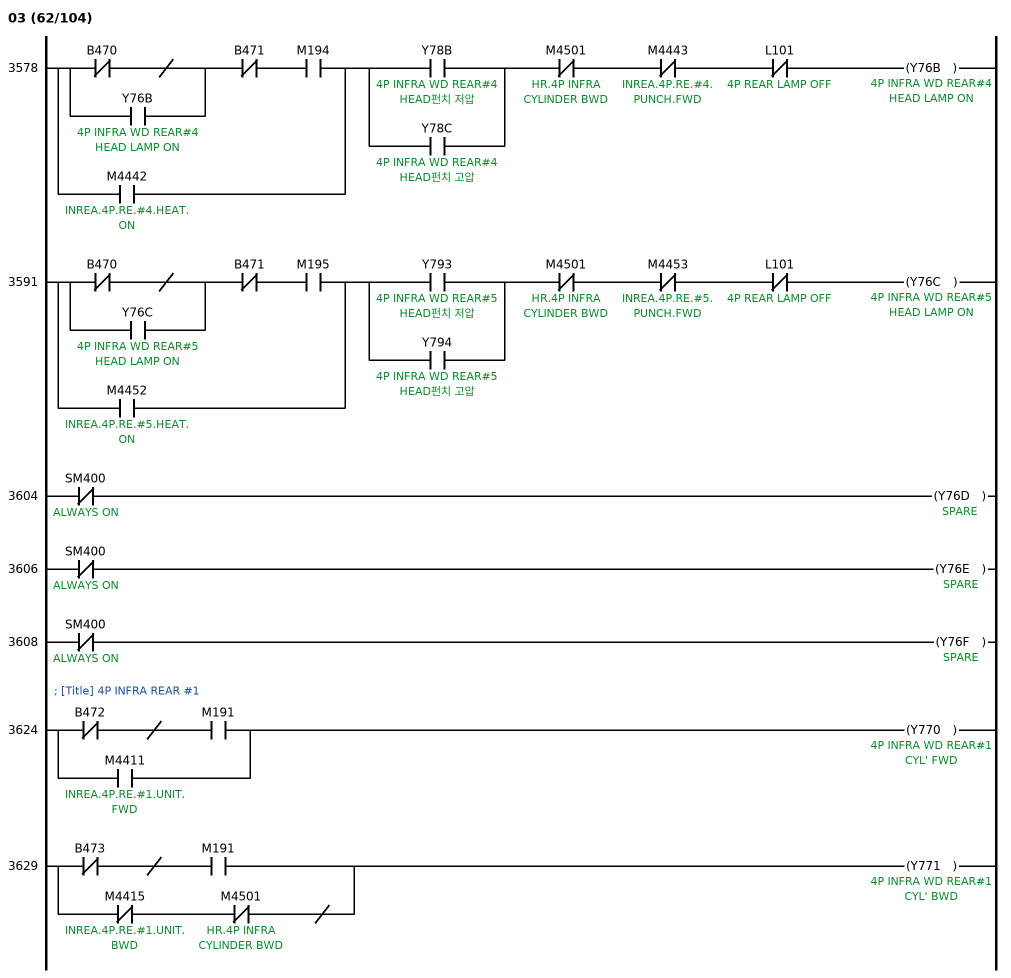
3578  LDI     B470
      INV
      OR      Y76B  ; 4P INFRA WD REAR#4 HEAD LAMP ON
      ANI     B471
      AND     M194
      OR      M4442  ; INREA.4P.RE.#4.HEAT.ON
      LD      Y78B  ; 4P INFRA WD REAR#4 HEAD펀치 저압
      OR      Y78C  ; 4P INFRA WD REAR#4 HEAD펀치 고압
      ANB
      ANI     M4501  ; HR.4P INFRA CYLINDER BWD
      ANI     M4443  ; INREA.4P.RE.#4.PUNCH.FWD
      ANI     L101  ; 4P REAR LAMP OFF
      OUT     Y76B  ; 4P INFRA WD REAR#4 HEAD LAMP ON
3591  LDI     B470
      INV
      OR      Y76C  ; 4P INFRA WD REAR#5 HEAD LAMP ON
      ANI     B471
      AND     M195
      OR      M4452  ; INREA.4P.RE.#5.HEAT.ON
      LD      Y793  ; 4P INFRA WD REAR#5 HEAD펀치 저압
      OR      Y794  ; 4P INFRA WD REAR#5 HEAD펀치 고압
      ANB
      ANI     M4501  ; HR.4P INFRA CYLINDER BWD
      ANI     M4453  ; INREA.4P.RE.#5.PUNCH.FWD
      ANI     L101  ; 4P REAR LAMP OFF
      OUT     Y76C  ; 4P INFRA WD REAR#5 HEAD LAMP ON
3604  LDI     SM400  ; ALWAYS ON
      OUT     Y76D  ; SPARE
3606  LDI     SM400  ; ALWAYS ON
      OUT     Y76E  ; SPARE
3608  LDI     SM400  ; ALWAYS ON
      OUT     Y76F  ; SPARE
; [Title] 4P INFRA REAR #1
3624  LDI     B472
      INV
      AND     M191
      OR      M4411  ; INREA.4P.RE.#1.UNIT.FWD
      OUT     Y770  ; 4P INFRA WD REAR#1 CYL' FWD
3629  LDI     B473
      INV
      AND     M191
      LDI     M4415  ; INREA.4P.RE.#1.UNIT.BWD
      ANI     M4501  ; HR.4P INFRA CYLINDER BWD
      INV
      ORB
      OUT     Y771  ; 4P INFRA WD REAR#1 CYL' BWD
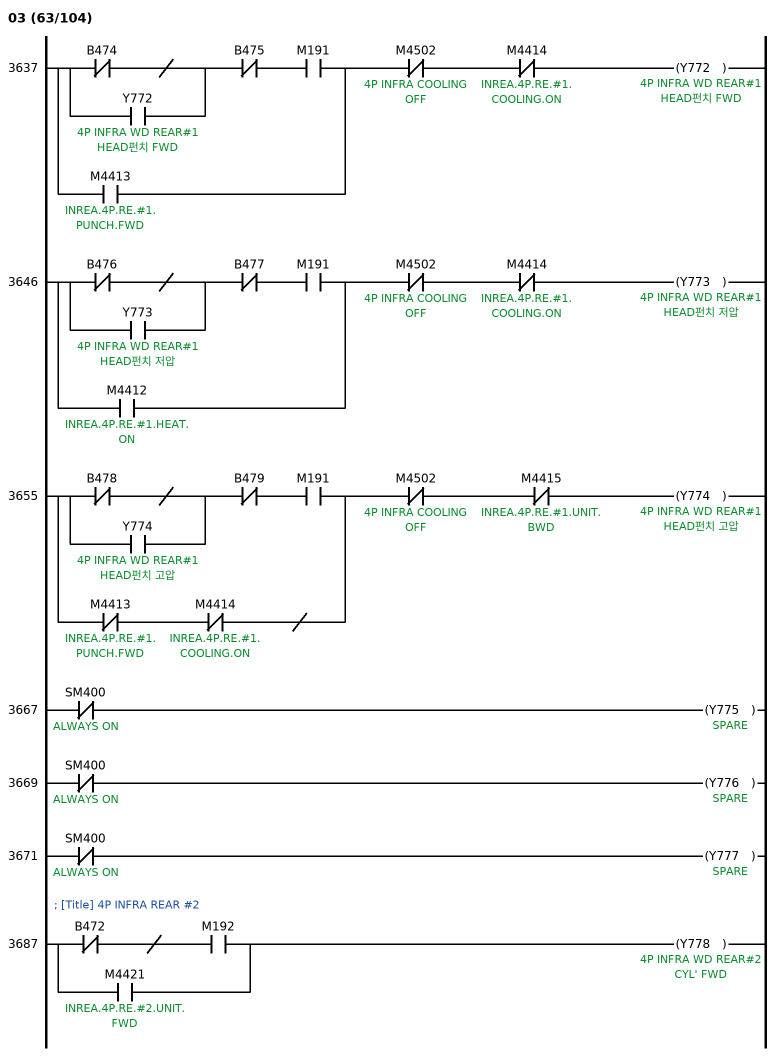
3637  LDI     B474
      INV
      OR      Y772  ; 4P INFRA WD REAR#1 HEAD펀치 FWD
      ANI     B475
      AND     M191
      OR      M4413  ; INREA.4P.RE.#1.PUNCH.FWD
      ANI     M4502  ; 4P INFRA COOLING OFF
      ANI     M4414  ; INREA.4P.RE.#1.COOLING.ON
      OUT     Y772  ; 4P INFRA WD REAR#1 HEAD펀치 FWD
3646  LDI     B476
      INV
      OR      Y773  ; 4P INFRA WD REAR#1 HEAD펀치 저압
      ANI     B477
      AND     M191
      OR      M4412  ; INREA.4P.RE.#1.HEAT.ON
      ANI     M4502  ; 4P INFRA COOLING OFF
      ANI     M4414  ; INREA.4P.RE.#1.COOLING.ON
      OUT     Y773  ; 4P INFRA WD REAR#1 HEAD펀치 저압
3655  LDI     B478
      INV
      OR      Y774  ; 4P INFRA WD REAR#1 HEAD펀치 고압
      ANI     B479
      AND     M191
      LDI     M4413  ; INREA.4P.RE.#1.PUNCH.FWD
      ANI     M4414  ; INREA.4P.RE.#1.COOLING.ON
      INV
      ORB
      ANI     M4502  ; 4P INFRA COOLING OFF
      ANI     M4415  ; INREA.4P.RE.#1.UNIT.BWD
      OUT     Y774  ; 4P INFRA WD REAR#1 HEAD펀치 고압
3667  LDI     SM400  ; ALWAYS ON
      OUT     Y775  ; SPARE
3669  LDI     SM400  ; ALWAYS ON
      OUT     Y776  ; SPARE
3671  LDI     SM400  ; ALWAYS ON
      OUT     Y777  ; SPARE
; [Title] 4P INFRA REAR #2
3687  LDI     B472
      INV
      AND     M192
      OR      M4421  ; INREA.4P.RE.#2.UNIT.FWD
      OUT     Y778  ; 4P INFRA WD REAR#2 CYL' FWD
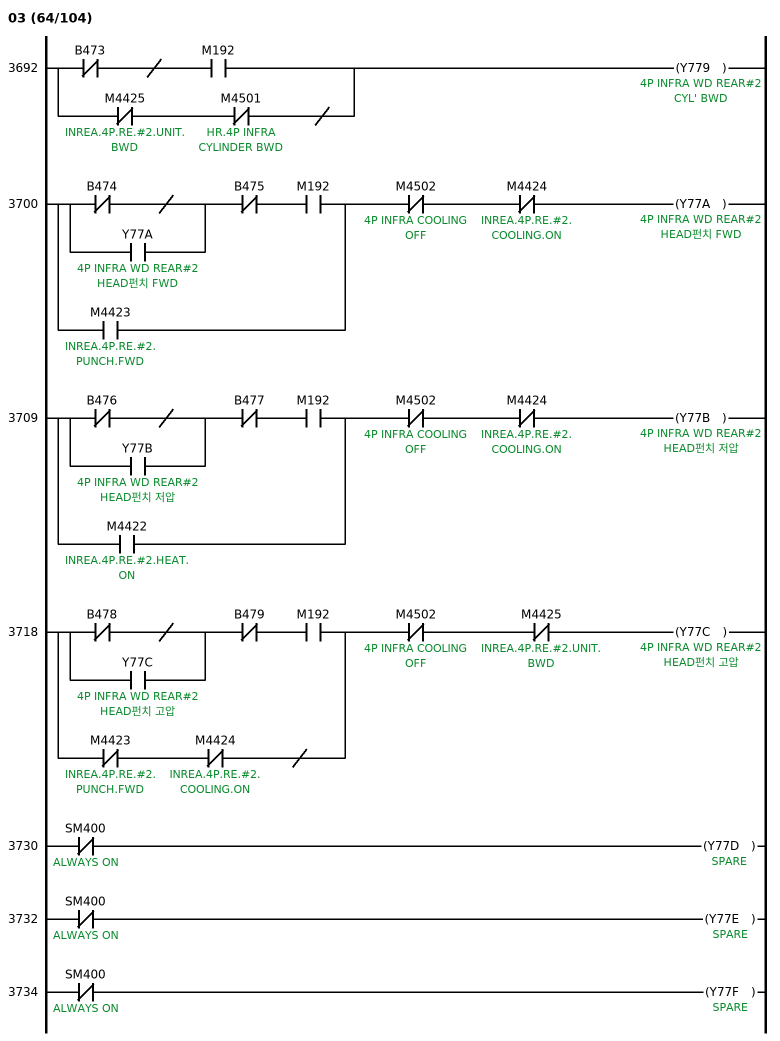
3692  LDI     B473
      INV
      AND     M192
      LDI     M4425  ; INREA.4P.RE.#2.UNIT.BWD
      ANI     M4501  ; HR.4P INFRA CYLINDER BWD
      INV
      ORB
      OUT     Y779  ; 4P INFRA WD REAR#2 CYL' BWD
3700  LDI     B474
      INV
      OR      Y77A  ; 4P INFRA WD REAR#2 HEAD펀치 FWD
      ANI     B475
      AND     M192
      OR      M4423  ; INREA.4P.RE.#2.PUNCH.FWD
      ANI     M4502  ; 4P INFRA COOLING OFF
      ANI     M4424  ; INREA.4P.RE.#2.COOLING.ON
      OUT     Y77A  ; 4P INFRA WD REAR#2 HEAD펀치 FWD
3709  LDI     B476
      INV
      OR      Y77B  ; 4P INFRA WD REAR#2 HEAD펀치 저압
      ANI     B477
      AND     M192
      OR      M4422  ; INREA.4P.RE.#2.HEAT.ON
      ANI     M4502  ; 4P INFRA COOLING OFF
      ANI     M4424  ; INREA.4P.RE.#2.COOLING.ON
      OUT     Y77B  ; 4P INFRA WD REAR#2 HEAD펀치 저압
3718  LDI     B478
      INV
      OR      Y77C  ; 4P INFRA WD REAR#2 HEAD펀치 고압
      ANI     B479
      AND     M192
      LDI     M4423  ; INREA.4P.RE.#2.PUNCH.FWD
      ANI     M4424  ; INREA.4P.RE.#2.COOLING.ON
      INV
      ORB
      ANI     M4502  ; 4P INFRA COOLING OFF
      ANI     M4425  ; INREA.4P.RE.#2.UNIT.BWD
      OUT     Y77C  ; 4P INFRA WD REAR#2 HEAD펀치 고압
3730  LDI     SM400  ; ALWAYS ON
      OUT     Y77D  ; SPARE
3732  LDI     SM400  ; ALWAYS ON
      OUT     Y77E  ; SPARE
3734  LDI     SM400  ; ALWAYS ON
      OUT     Y77F  ; SPARE
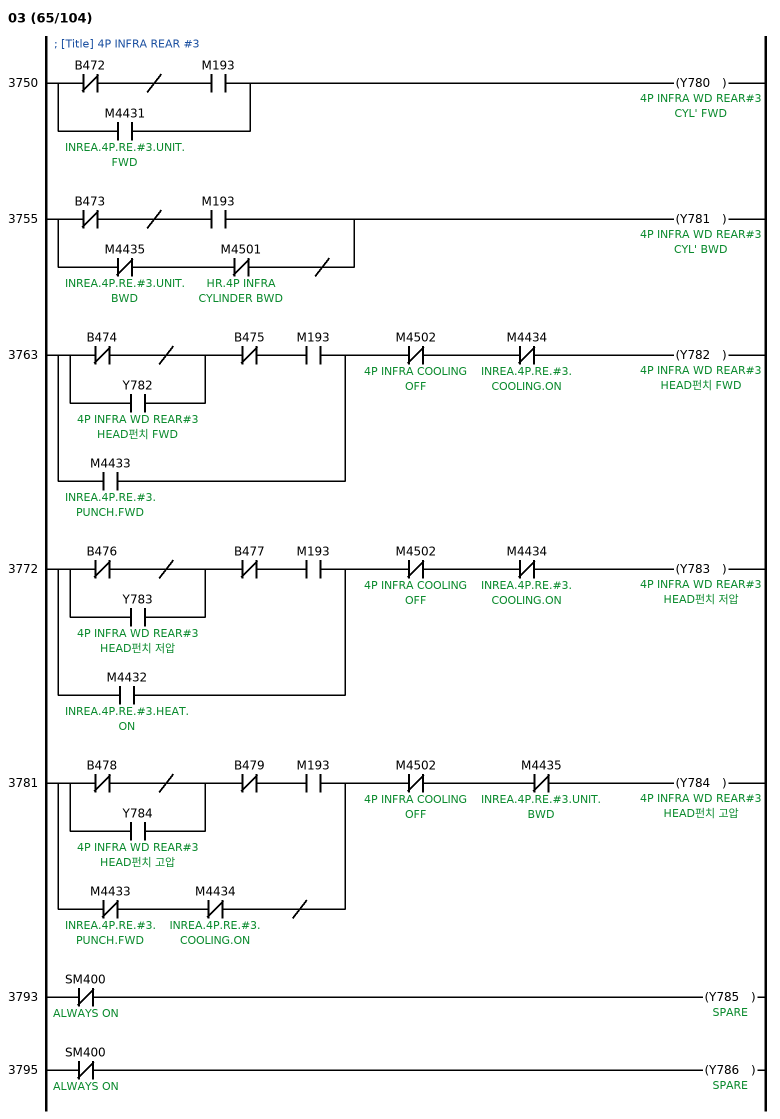
; [Title] 4P INFRA REAR #3
3750  LDI     B472
      INV
      AND     M193
      OR      M4431  ; INREA.4P.RE.#3.UNIT.FWD
      OUT     Y780  ; 4P INFRA WD REAR#3 CYL' FWD
3755  LDI     B473
      INV
      AND     M193
      LDI     M4435  ; INREA.4P.RE.#3.UNIT.BWD
      ANI     M4501  ; HR.4P INFRA CYLINDER BWD
      INV
      ORB
      OUT     Y781  ; 4P INFRA WD REAR#3 CYL' BWD
3763  LDI     B474
      INV
      OR      Y782  ; 4P INFRA WD REAR#3 HEAD펀치 FWD
      ANI     B475
      AND     M193
      OR      M4433  ; INREA.4P.RE.#3.PUNCH.FWD
      ANI     M4502  ; 4P INFRA COOLING OFF
      ANI     M4434  ; INREA.4P.RE.#3.COOLING.ON
      OUT     Y782  ; 4P INFRA WD REAR#3 HEAD펀치 FWD
3772  LDI     B476
      INV
      OR      Y783  ; 4P INFRA WD REAR#3 HEAD펀치 저압
      ANI     B477
      AND     M193
      OR      M4432  ; INREA.4P.RE.#3.HEAT.ON
      ANI     M4502  ; 4P INFRA COOLING OFF
      ANI     M4434  ; INREA.4P.RE.#3.COOLING.ON
      OUT     Y783  ; 4P INFRA WD REAR#3 HEAD펀치 저압
3781  LDI     B478
      INV
      OR      Y784  ; 4P INFRA WD REAR#3 HEAD펀치 고압
      ANI     B479
      AND     M193
      LDI     M4433  ; INREA.4P.RE.#3.PUNCH.FWD
      ANI     M4434  ; INREA.4P.RE.#3.COOLING.ON
      INV
      ORB
      ANI     M4502  ; 4P INFRA COOLING OFF
      ANI     M4435  ; INREA.4P.RE.#3.UNIT.BWD
      OUT     Y784  ; 4P INFRA WD REAR#3 HEAD펀치 고압
3793  LDI     SM400  ; ALWAYS ON
      OUT     Y785  ; SPARE
3795  LDI     SM400  ; ALWAYS ON
      OUT     Y786  ; SPARE
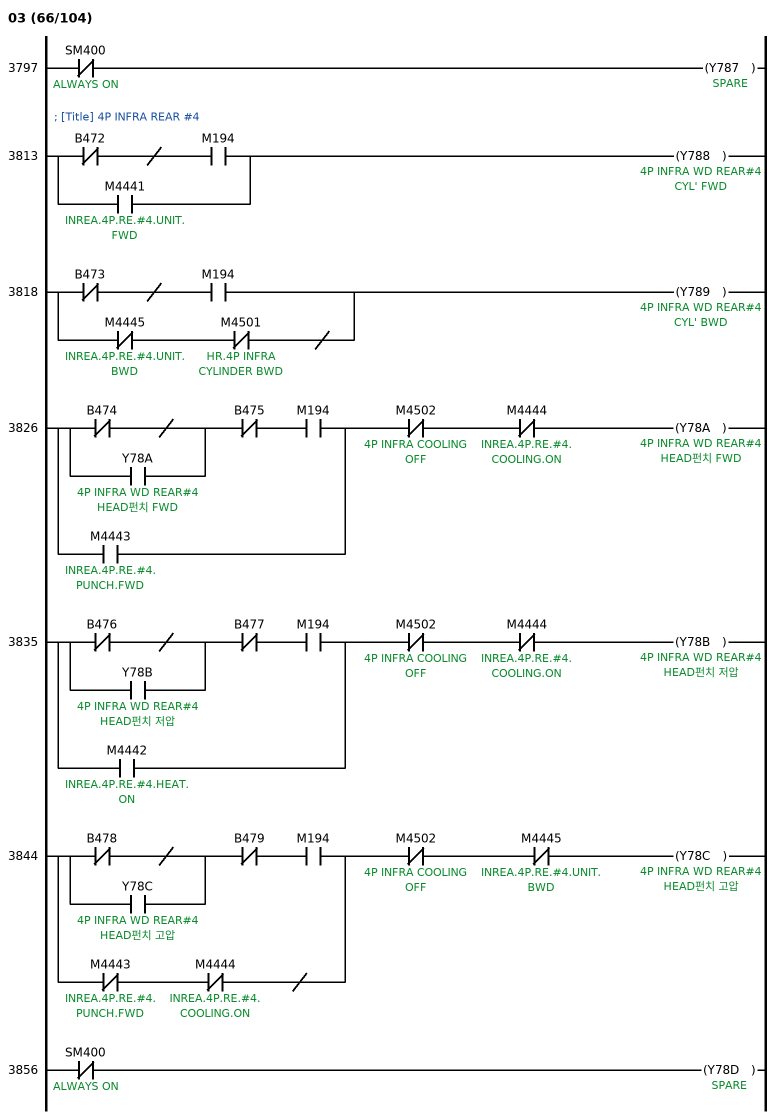
3797  LDI     SM400  ; ALWAYS ON
      OUT     Y787  ; SPARE
; [Title] 4P INFRA REAR #4
3813  LDI     B472
      INV
      AND     M194
      OR      M4441  ; INREA.4P.RE.#4.UNIT.FWD
      OUT     Y788  ; 4P INFRA WD REAR#4 CYL' FWD
3818  LDI     B473
      INV
      AND     M194
      LDI     M4445  ; INREA.4P.RE.#4.UNIT.BWD
      ANI     M4501  ; HR.4P INFRA CYLINDER BWD
      INV
      ORB
      OUT     Y789  ; 4P INFRA WD REAR#4 CYL' BWD
3826  LDI     B474
      INV
      OR      Y78A  ; 4P INFRA WD REAR#4 HEAD펀치 FWD
      ANI     B475
      AND     M194
      OR      M4443  ; INREA.4P.RE.#4.PUNCH.FWD
      ANI     M4502  ; 4P INFRA COOLING OFF
      ANI     M4444  ; INREA.4P.RE.#4.COOLING.ON
      OUT     Y78A  ; 4P INFRA WD REAR#4 HEAD펀치 FWD
3835  LDI     B476
      INV
      OR      Y78B  ; 4P INFRA WD REAR#4 HEAD펀치 저압
      ANI     B477
      AND     M194
      OR      M4442  ; INREA.4P.RE.#4.HEAT.ON
      ANI     M4502  ; 4P INFRA COOLING OFF
      ANI     M4444  ; INREA.4P.RE.#4.COOLING.ON
      OUT     Y78B  ; 4P INFRA WD REAR#4 HEAD펀치 저압
3844  LDI     B478
      INV
      OR      Y78C  ; 4P INFRA WD REAR#4 HEAD펀치 고압
      ANI     B479
      AND     M194
      LDI     M4443  ; INREA.4P.RE.#4.PUNCH.FWD
      ANI     M4444  ; INREA.4P.RE.#4.COOLING.ON
      INV
      ORB
      ANI     M4502  ; 4P INFRA COOLING OFF
      ANI     M4445  ; INREA.4P.RE.#4.UNIT.BWD
      OUT     Y78C  ; 4P INFRA WD REAR#4 HEAD펀치 고압
3856  LDI     SM400  ; ALWAYS ON
      OUT     Y78D  ; SPARE
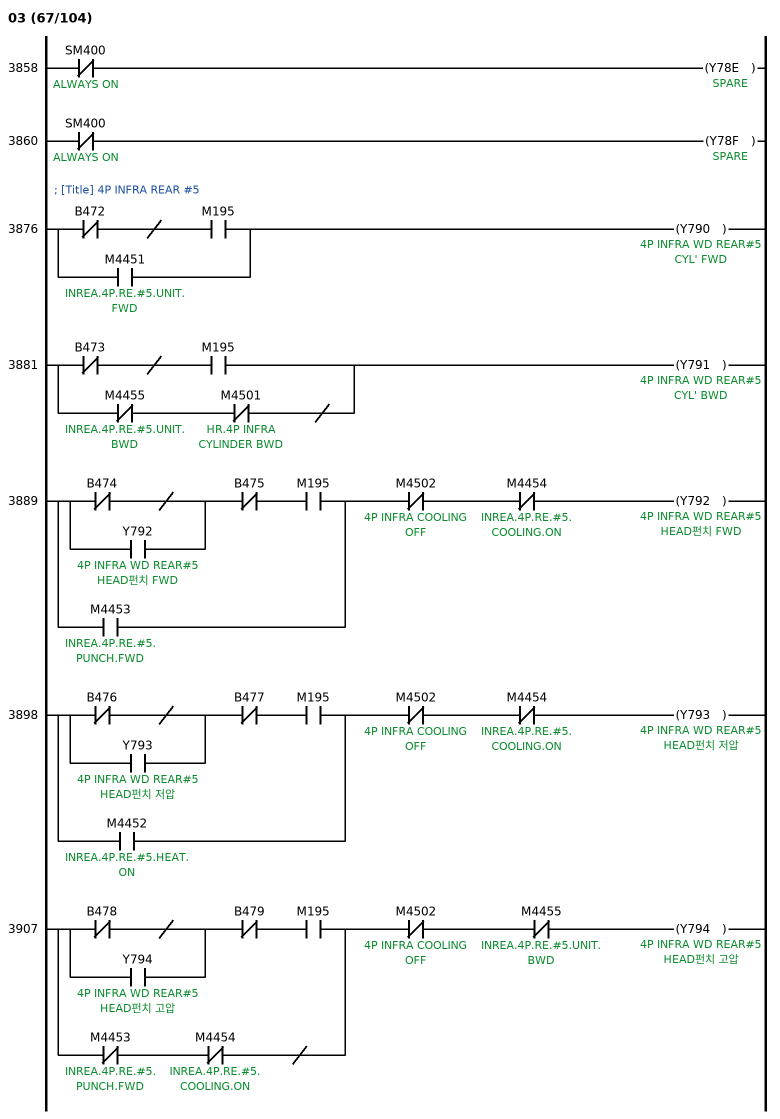
3858  LDI     SM400  ; ALWAYS ON
      OUT     Y78E  ; SPARE
3860  LDI     SM400  ; ALWAYS ON
      OUT     Y78F  ; SPARE
; [Title] 4P INFRA REAR #5
3876  LDI     B472
      INV
      AND     M195
      OR      M4451  ; INREA.4P.RE.#5.UNIT.FWD
      OUT     Y790  ; 4P INFRA WD REAR#5 CYL' FWD
3881  LDI     B473
      INV
      AND     M195
      LDI     M4455  ; INREA.4P.RE.#5.UNIT.BWD
      ANI     M4501  ; HR.4P INFRA CYLINDER BWD
      INV
      ORB
      OUT     Y791  ; 4P INFRA WD REAR#5 CYL' BWD
3889  LDI     B474
      INV
      OR      Y792  ; 4P INFRA WD REAR#5 HEAD펀치 FWD
      ANI     B475
      AND     M195
      OR      M4453  ; INREA.4P.RE.#5.PUNCH.FWD
      ANI     M4502  ; 4P INFRA COOLING OFF
      ANI     M4454  ; INREA.4P.RE.#5.COOLING.ON
      OUT     Y792  ; 4P INFRA WD REAR#5 HEAD펀치 FWD
3898  LDI     B476
      INV
      OR      Y793  ; 4P INFRA WD REAR#5 HEAD펀치 저압
      ANI     B477
      AND     M195
      OR      M4452  ; INREA.4P.RE.#5.HEAT.ON
      ANI     M4502  ; 4P INFRA COOLING OFF
      ANI     M4454  ; INREA.4P.RE.#5.COOLING.ON
      OUT     Y793  ; 4P INFRA WD REAR#5 HEAD펀치 저압
3907  LDI     B478
      INV
      OR      Y794  ; 4P INFRA WD REAR#5 HEAD펀치 고압
      ANI     B479
      AND     M195
      LDI     M4453  ; INREA.4P.RE.#5.PUNCH.FWD
      ANI     M4454  ; INREA.4P.RE.#5.COOLING.ON
      INV
      ORB
      ANI     M4502  ; 4P INFRA COOLING OFF
      ANI     M4455  ; INREA.4P.RE.#5.UNIT.BWD
      OUT     Y794  ; 4P INFRA WD REAR#5 HEAD펀치 고압
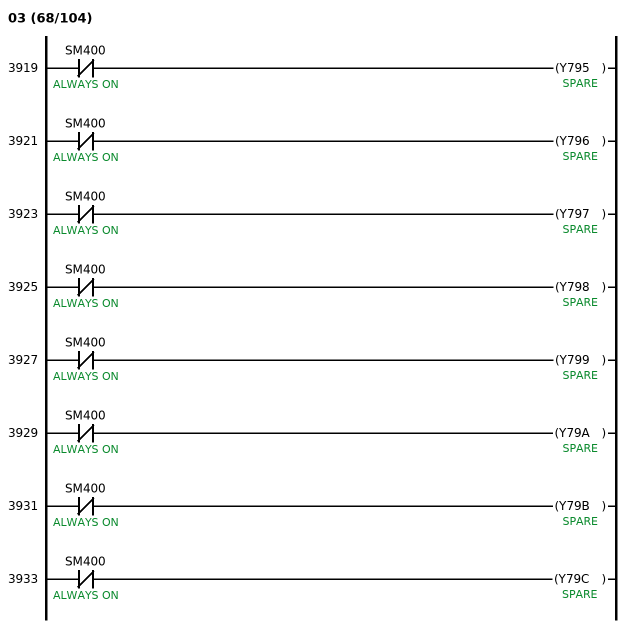
3919  LDI     SM400  ; ALWAYS ON
      OUT     Y795  ; SPARE
3921  LDI     SM400  ; ALWAYS ON
      OUT     Y796  ; SPARE
3923  LDI     SM400  ; ALWAYS ON
      OUT     Y797  ; SPARE
3925  LDI     SM400  ; ALWAYS ON
      OUT     Y798  ; SPARE
3927  LDI     SM400  ; ALWAYS ON
      OUT     Y799  ; SPARE
3929  LDI     SM400  ; ALWAYS ON
      OUT     Y79A  ; SPARE
3931  LDI     SM400  ; ALWAYS ON
      OUT     Y79B  ; SPARE
3933  LDI     SM400  ; ALWAYS ON
      OUT     Y79C  ; SPARE
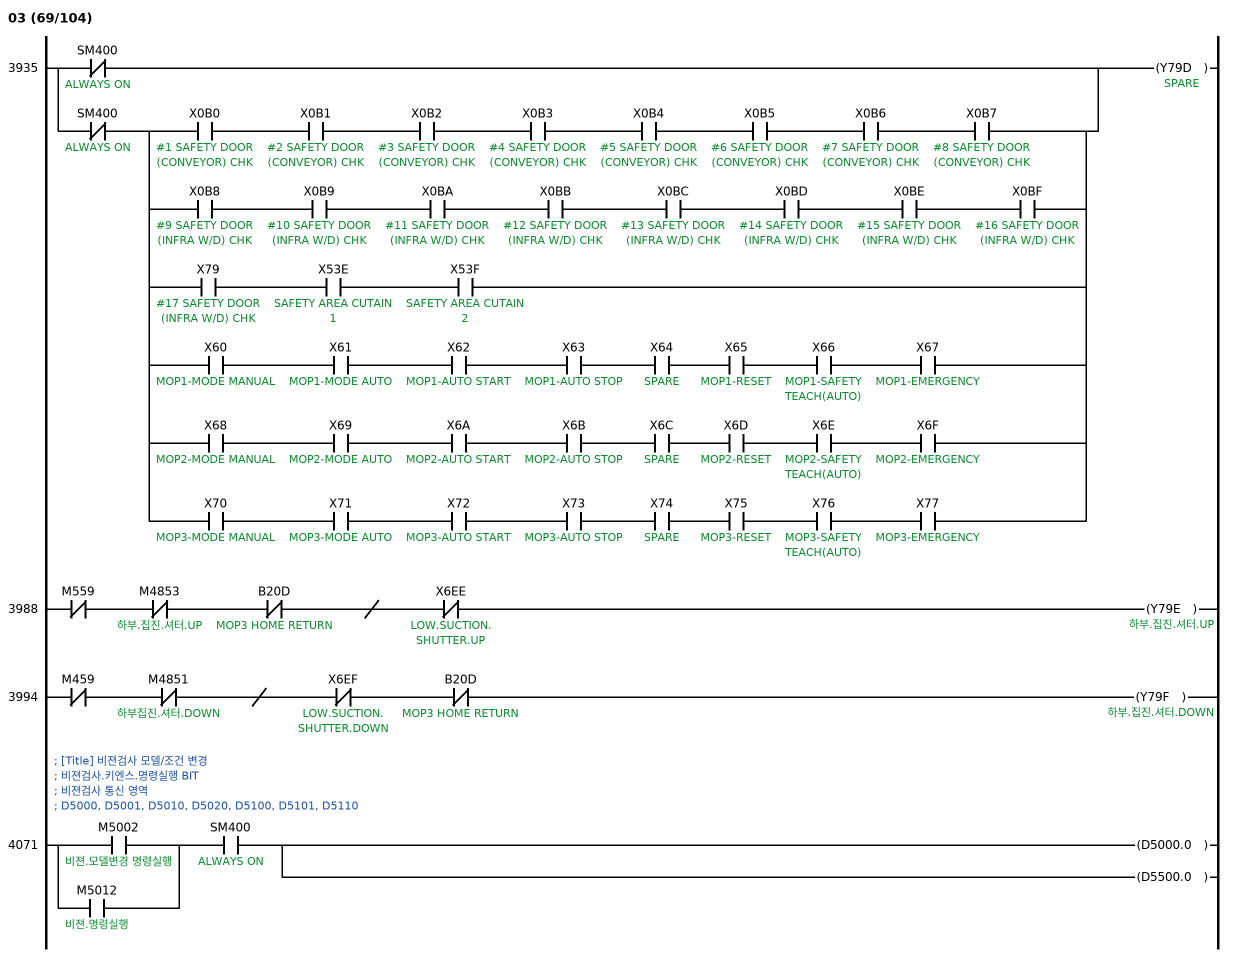
3935  LDI     SM400  ; ALWAYS ON
      LDI     SM400  ; ALWAYS ON
      LD      X0B0  ; #1 SAFETY DOOR (CONVEYOR) CHK
      AND     X0B1  ; #2 SAFETY DOOR (CONVEYOR) CHK
      AND     X0B2  ; #3 SAFETY DOOR (CONVEYOR) CHK
      AND     X0B3  ; #4 SAFETY DOOR (CONVEYOR) CHK
      AND     X0B4  ; #5 SAFETY DOOR (CONVEYOR) CHK
      AND     X0B5  ; #6 SAFETY DOOR (CONVEYOR) CHK
      AND     X0B6  ; #7 SAFETY DOOR (CONVEYOR) CHK
      AND     X0B7  ; #8 SAFETY DOOR (CONVEYOR) CHK
      LD      X0B8  ; #9 SAFETY DOOR (INFRA W/D) CHK
      AND     X0B9  ; #10 SAFETY DOOR (INFRA W/D) CHK
      AND     X0BA  ; #11 SAFETY DOOR (INFRA W/D) CHK
      AND     X0BB  ; #12 SAFETY DOOR (INFRA W/D) CHK
      AND     X0BC  ; #13 SAFETY DOOR (INFRA W/D) CHK
      AND     X0BD  ; #14 SAFETY DOOR (INFRA W/D) CHK
      AND     X0BE  ; #15 SAFETY DOOR (INFRA W/D) CHK
      AND     X0BF  ; #16 SAFETY DOOR (INFRA W/D) CHK
      ORB
      LD      X79  ; #17 SAFETY DOOR (INFRA W/D) CHK
      AND     X53E  ; SAFETY AREA CUTAIN 1
      AND     X53F  ; SAFETY AREA CUTAIN 2
      ORB
      LD      X60  ; MOP1-MODE MANUAL
      AND     X61  ; MOP1-MODE AUTO
      AND     X62  ; MOP1-AUTO START
      AND     X63  ; MOP1-AUTO STOP
      AND     X64  ; SPARE
      AND     X65  ; MOP1-RESET
      AND     X66  ; MOP1-SAFETY TEACH(AUTO)
      AND     X67  ; MOP1-EMERGENCY
      ORB
      LD      X68  ; MOP2-MODE MANUAL
      AND     X69  ; MOP2-MODE AUTO
      AND     X6A  ; MOP2-AUTO START
      AND     X6B  ; MOP2-AUTO STOP
      AND     X6C  ; SPARE
      AND     X6D  ; MOP2-RESET
      AND     X6E  ; MOP2-SAFETY TEACH(AUTO)
      AND     X6F  ; MOP2-EMERGENCY
      ORB
      LD      X70  ; MOP3-MODE MANUAL
      AND     X71  ; MOP3-MODE AUTO
      AND     X72  ; MOP3-AUTO START
      AND     X73  ; MOP3-AUTO STOP
      AND     X74  ; SPARE
      AND     X75  ; MOP3-RESET
      AND     X76  ; MOP3-SAFETY TEACH(AUTO)
      AND     X77  ; MOP3-EMERGENCY
      ORB
      ANB
      ORB
      OUT     Y79D  ; SPARE
3988  LDI     M559
      ANI     M4853  ; 하부.집진.셔터.UP
      ANI     B20D  ; MOP3 HOME RETURN
      INV
      ANI     X6EE  ; LOW.SUCTION.SHUTTER.UP
      OUT     Y79E  ; 하부.집진.셔터.UP
3994  LDI     M459
      ANI     M4851  ; 하부집진.셔터.DOWN
      INV
      ANI     X6EF  ; LOW.SUCTION.SHUTTER.DOWN
      ANI     B20D  ; MOP3 HOME RETURN
      OUT     Y79F  ; 하부.집진.셔터.DOWN
; [Title] 비젼검사 모델/조건 변경
; 비젼검사.키엔스.명령실행 BIT
; 비젼검사 통신 영역
; D5000, D5001, D5010, D5020, D5100, D5101, D5110
4071  LD      M5002  ; 비젼.모델변경 명령실행
      OR      M5012  ; 비젼.명령실행
      AND     SM400  ; ALWAYS ON
      OUT     D5000.0
      OUT     D5500.0
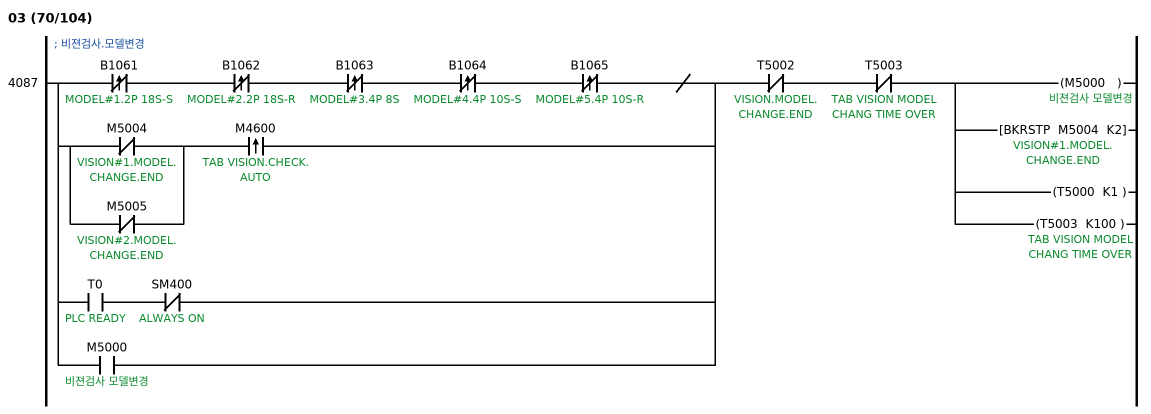
; 비젼검사.모델변경
4087  LDPI    B1061  ; MODEL#1.2P 18S-S
      ANDPI   B1062  ; MODEL#2.2P 18S-R
      ANDPI   B1063  ; MODEL#3.4P 8S
      ANDPI   B1064  ; MODEL#4.4P 10S-S
      ANDPI   B1065  ; MODEL#5.4P 10S-R
      INV
      LDI     M5004  ; VISION#1.MODEL.CHANGE.END
      ORI     M5005  ; VISION#2.MODEL.CHANGE.END
      ANDP    M4600  ; TAB VISION.CHECK.AUTO
      ORB
      LD      T0  ; PLC READY
      ANI     SM400  ; ALWAYS ON
      ORB
      OR      M5000  ; 비젼검사 모델변경
      ANI     T5002  ; VISION.MODEL.CHANGE.END
      ANI     T5003  ; TAB VISION MODEL CHANG TIME OVER
      OUT     M5000  ; 비젼검사 모델변경
      BKRSTP  M5004 K2
      OUT     T5000 K1
      OUT     T5003 K100  ; TAB VISION MODEL CHANG TIME OVER
